KUKA KRL program: EPS_2_251349_MH87A_A_20250929014658.src

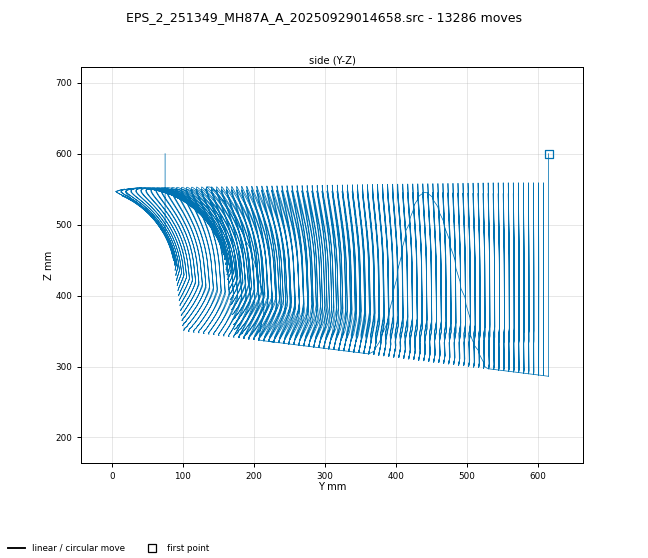
[picture p0: tool path of EPS_2_251349_MH87A_A_20250929014658.src, 13286 of 13288 moves have a stored position in this frame; points joined in program order, loops and branches not executed]
&ACCESS RVP
&REL 4
&COMMENT QRS 19112012
&PARAM EDITMASK = *
DEF PART()
EXT BAS (BAS_COMMAND :IN,REAL :IN )
INT I
BAS (#INITMOV,0 )

;KUKA QRS Post kuka4.cps  Date:22-06-2017 !

File_ID=2862

QRS_PRE_INIT()

;Init var - Until changes are made in qrs_pre_init
Outlet_Square_prg=0
Inlet_1_Square_prg=0
Inlet_2_Square_prg=0
Inlet_3_Square_prg=0
Inlet_4_Square_prg=0
Inlet_5_Square_prg=0

Outlet_1={X 0.000, Y 535.490, Z 458.500, B 0.000, E1 0.000 }
Inlet_1={X 0.000, Y 536.560, Z 443.500, B 0.000, E1 156.000 }
Outlet_1_type=201
Inlet_1_type=201
;QRS#1=Sidecore dimensions
;QRS#2=200-8" PVC SDR 35
;QRS#3=200-8" PVC SDR 35
;QRS#4=
;QRS#5=
;QRS#6=
;QRS#7=
;QRS#8=
;QRS#9=12-08 PSX
;QRS#10=12-08 PSX
;QRS#11=
;QRS#12=
;QRS#13=
;QRS#14=
;QRS#15=
;QRS#16=1220x127x838 2,75'
;QRS#17=EPS Height
;QRS#18=559
;QRS#19=*
;QRS#20= UPDATED VERSION 22-06-2017
;QRS#21=*
Outlet_Square=0100
Inlet_1_Square=0100
Inlet_2_Square=0
Inlet_3_Square=0
Inlet_4_Square=0
Inlet_5_Square=0
Mill_Square=1
Outlet_Square_Prg=204
Inlet_1_Square_prg=204

QRS_INIT()

$ADVANCE=5

; T1
PTP {E1 173.604,E2 173.604}
PTP {X 0,Y 615.51,A -85,B 0,C 180,E1 173.604,E2 173.604,E3 0,E4 0,E5 0,E6 0}
QRS_SPEED_INIT()
LIN {X 0,Y 615.51,Z 600,A -85,B 0,C 180,E1 173.604,E2 173.604,E3 0,E4 0,E5 0,E6 0} C_VEL
LIN {X 0,Y 615.51,Z 296.361,A -85,B 0,C 180,E1 173.604,E2 173.604} C_VEL
LIN {X 0,Y 615.51,Z 288.184,A -85,B 0,C 180,E1 173.604,E2 173.604} C_VEL
LIN {X 0,Y 615.494,Z 286.184,A -85,B 0,C 180,E1 173.418,E2 173.418} C_VEL
LIN {X 0,Y 615.499,Z 286.199,A -85,B 0,C 180,E1 170.801,E2 170.801} C_VEL
LIN {X 0,Y 615.469,Z 286.19,A -85,B 0,C 180,E1 168.139,E2 168.139} C_VEL
LIN {X 0,Y 615.478,Z 286.181,A -85,B 0,C 180,E1 165.451,E2 165.451} C_VEL
LIN {X 0,Y 615.488,Z 286.183,A -85,B 0,C 180,E1 162.729,E2 162.729} C_VEL
LIN {X 0,Y 615.491,Z 286.202,A -85,B 0,C 180,E1 159.967,E2 159.967} C_VEL
LIN {X 0,Y 615.48,Z 286.198,A -85,B 0,C 180,E1 157.656,E2 157.656} C_VEL
LIN {X 0,Y 615.46,Z 286.188,A -85,B 0,C 180,E1 155.007,E2 155.007} C_VEL
LIN {X 0,Y 615.459,Z 286.188,A -85,B 0,C 180,E1 152.821,E2 152.821} C_VEL
LIN {X 0,Y 615.478,Z 286.181,A -85,B 0,C 180,E1 150.207,E2 150.207} C_VEL
LIN {X 0,Y 615.487,Z 286.186,A -85,B 0,C 180,E1 147.542,E2 147.542} C_VEL
LIN {X 0,Y 615.487,Z 286.192,A -85,B 0,C 180,E1 145.185,E2 145.185} C_VEL
LIN {X 0,Y 615.491,Z 286.201,A -85,B 0,C 180,E1 142.758,E2 142.758} C_VEL
LIN {X 0,Y 615.474,Z 286.193,A -85,B 0,C 180,E1 140.249,E2 140.249} C_VEL
LIN {X 0,Y 615.456,Z 286.187,A -85,B 0,C 180,E1 137.644,E2 137.644} C_VEL
LIN {X 0,Y 615.473,Z 286.183,A -85,B 0,C 180,E1 134.93,E2 134.93} C_VEL
LIN {X 0,Y 615.498,Z 286.371,A -85,B 0,C 180,E1 134.036,E2 134.036} C_VEL
LIN {X 0,Y 615.487,Z 302.509,A -85,B 0,C 180,E1 131.474,E2 131.474} C_VEL
LIN {X 0,Y 615.461,Z 320.425,A -85,B 0,C 180,E1 128.697,E2 128.697} C_VEL
LIN {X 0,Y 615.464,Z 332.446,A -85,B 0,C 180,E1 126.871,E2 126.871} C_VEL
LIN {X 0,Y 615.462,Z 333.679,A -85,B 0,C 180,E1 126.807,E2 126.807} C_VEL
LIN {X 0,Y 615.496,Z 437.942,A -85,B 0,C 180,E1 125.565,E2 125.565} C_VEL
LIN {X 0,Y 615.494,Z 448.449,A -85,B 0,C 180,E1 125.364,E2 125.364} C_VEL
LIN {X 0,Y 615.497,Z 459.189,A -85,B 0,C 180,E1 125.064,E2 125.064} C_VEL
LIN {X 0,Y 615.499,Z 468.978,A -85,B 0,C 180,E1 124.702,E2 124.702} C_VEL
LIN {X 0,Y 615.478,Z 479.707,A -85,B 0,C 180,E1 124.192,E2 124.192} C_VEL
LIN {X 0,Y 615.49,Z 488.871,A -85,B 0,C 180,E1 123.656,E2 123.656} C_VEL
LIN {X 0,Y 615.499,Z 498.772,A -85,B 0,C 180,E1 122.943,E2 122.943} C_VEL
LIN {X 0,Y 615.495,Z 505.946,A -85,B 0,C 180,E1 122.332,E2 122.332} C_VEL
LIN {X 0,Y 615.494,Z 513.767,A -85,B 0,C 180,E1 121.535,E2 121.535} C_VEL
LIN {X 0,Y 615.497,Z 520.403,A -85,B 0,C 180,E1 120.729,E2 120.729} C_VEL
LIN {X 0,Y 615.486,Z 526.732,A -85,B 0,C 180,E1 119.794,E2 119.794} C_VEL
LIN {X 0,Y 615.492,Z 531.077,A -85,B 0,C 180,E1 119.031,E2 119.031} C_VEL
LIN {X 0,Y 615.49,Z 535.996,A -85,B 0,C 180,E1 117.915,E2 117.915} C_VEL
LIN {X 0,Y 615.486,Z 538.972,A -85,B 0,C 180,E1 117.045,E2 117.045} C_VEL
LIN {X 0,Y 615.495,Z 542.092,A -85,B 0,C 180,E1 115.57,E2 115.57} C_VEL
LIN {X 0,Y 615.495,Z 542.897,A -85,B 0,C 180,E1 114.991,E2 114.991} C_VEL
LIN {X 0,Y 615.493,Z 543.382,A -85,B 0,C 180,E1 114.009,E2 114.009} C_VEL
LIN {X 0,Y 615.485,Z 542.815,A -85,B 0,C 180,E1 112.845,E2 112.845} C_VEL
LIN {X 0,Y 615.496,Z 541.803,A -85,B 0,C 180,E1 112.136,E2 112.136} C_VEL
LIN {X 0,Y 615.491,Z 538.547,A -85,B 0,C 180,E1 110.731,E2 110.731} C_VEL
LIN {X 0,Y 615.49,Z 534.776,A -85,B 0,C 180,E1 109.685,E2 109.685} C_VEL
LIN {X 0,Y 615.496,Z 529.572,A -85,B 0,C 180,E1 108.607,E2 108.607} C_VEL
LIN {X 0,Y 615.491,Z 524.695,A -85,B 0,C 180,E1 107.785,E2 107.785} C_VEL
LIN {X 0,Y 615.493,Z 517.044,A -85,B 0,C 180,E1 106.757,E2 106.757} C_VEL
LIN {X 0,Y 615.5,Z 510.634,A -85,B 0,C 180,E1 106.037,E2 106.037} C_VEL
LIN {X 0,Y 615.497,Z 501.923,A -85,B 0,C 180,E1 105.226,E2 105.226} C_VEL
LIN {X 0,Y 615.49,Z 493.177,A -85,B 0,C 180,E1 104.549,E2 104.549} C_VEL
LIN {X 0,Y 615.487,Z 484.879,A -85,B 0,C 180,E1 104.008,E2 104.008} C_VEL
LIN {X 0,Y 615.485,Z 474.438,A -85,B 0,C 180,E1 103.453,E2 103.453} C_VEL
LIN {X 0,Y 615.498,Z 464.571,A -85,B 0,C 180,E1 103.033,E2 103.033} C_VEL
LIN {X 0,Y 615.498,Z 454.476,A -85,B 0,C 180,E1 102.697,E2 102.697} C_VEL
LIN {X 0,Y 615.497,Z 442.926,A -85,B 0,C 180,E1 102.425,E2 102.425} C_VEL
LIN {X 0,Y 615.497,Z 424.681,A -85,B 0,C 180,E1 102.174,E2 102.174} C_VEL
LIN {X 0,Y 615.49,Z 333.446,A -85,B 0,C 180,E1 101.098,E2 101.098} C_VEL
LIN {X 0,Y 615.491,Z 332.123,A -85,B 0,C 180,E1 101.003,E2 101.003} C_VEL
LIN {X 0,Y 615.474,Z 314.962,A -85,B 0,C 180,E1 98.371,E2 98.371} C_VEL
LIN {X 0,Y 615.488,Z 296.979,A -85,B 0,C 180,E1 95.57,E2 95.57} C_VEL
LIN {X 0,Y 615.497,Z 286.302,A -85,B 0,C 180,E1 93.846,E2 93.846} C_VEL
LIN {X 0,Y 615.493,Z 286.19,A -85,B 0,C 180,E1 91.309,E2 91.309} C_VEL
LIN {X 0,Y 615.478,Z 286.183,A -85,B 0,C 180,E1 88.691,E2 88.691} C_VEL
LIN {X 0,Y 615.472,Z 286.181,A -85,B 0,C 180,E1 86.071,E2 86.071} C_VEL
LIN {X 0,Y 615.49,Z 286.183,A -85,B 0,C 180,E1 83.42,E2 83.42} C_VEL
LIN {X 0,Y 615.494,Z 286.195,A -85,B 0,C 180,E1 80.801,E2 80.801} C_VEL
LIN {X 0,Y 615.496,Z 286.188,A -85,B 0,C 180,E1 78.139,E2 78.139} C_VEL
LIN {X 0,Y 615.472,Z 286.183,A -85,B 0,C 180,E1 75.45,E2 75.45} C_VEL
LIN {X 0,Y 615.472,Z 286.182,A -85,B 0,C 180,E1 72.729,E2 72.729} C_VEL
LIN {X 0,Y 615.493,Z 286.191,A -85,B 0,C 180,E1 69.967,E2 69.967} C_VEL
LIN {X 0,Y 615.49,Z 286.189,A -85,B 0,C 180,E1 67.155,E2 67.155} C_VEL
LIN {X 0,Y 615.463,Z 286.184,A -85,B 0,C 180,E1 64.436,E2 64.436} C_VEL
LIN {X 0,Y 615.463,Z 286.183,A -85,B 0,C 180,E1 62.084,E2 62.084} C_VEL
LIN {X 0,Y 615.463,Z 286.183,A -85,B 0,C 180,E1 59.838,E2 59.838} C_VEL
LIN {X 0,Y 615.461,Z 286.184,A -85,B 0,C 180,E1 57.541,E2 57.541} C_VEL
LIN {X 0,Y 615.472,Z 286.183,A -85,B 0,C 180,E1 55.184,E2 55.184} C_VEL
LIN {X 0,Y 615.486,Z 286.183,A -85,B 0,C 180,E1 52.758,E2 52.758} C_VEL
LIN {X 0,Y 615.497,Z 286.198,A -85,B 0,C 180,E1 49.91,E2 49.91} C_VEL
LIN {X 0,Y 615.494,Z 286.196,A -85,B 0,C 180,E1 47.647,E2 47.647} C_VEL
LIN {X 0,Y 615.467,Z 286.186,A -85,B 0,C 180,E1 44.929,E2 44.929} C_VEL
LIN {X 0,Y 615.456,Z 286.185,A -85,B 0,C 180,E1 42.356,E2 42.356} C_VEL
LIN {X 0,Y 615.474,Z 286.183,A -85,B 0,C 180,E1 39.751,E2 39.751} C_VEL
LIN {X 0,Y 615.491,Z 286.197,A -85,B 0,C 180,E1 36.937,E2 36.937} C_VEL
LIN {X 0,Y 615.465,Z 286.188,A -85,B 0,C 180,E1 34.023,E2 34.023} C_VEL
LIN {X 0,Y 615.456,Z 286.187,A -85,B 0,C 180,E1 31.687,E2 31.687} C_VEL
LIN {X 0,Y 615.452,Z 286.187,A -85,B 0,C 180,E1 29.408,E2 29.408} C_VEL
LIN {X 0,Y 615.45,Z 286.186,A -85,B 0,C 180,E1 27.038,E2 27.038} C_VEL
LIN {X 0,Y 615.448,Z 286.188,A -85,B 0,C 180,E1 24.994,E2 24.994} C_VEL
LIN {X 0,Y 615.449,Z 286.188,A -85,B 0,C 180,E1 22.846,E2 22.846} C_VEL
LIN {X 0,Y 615.447,Z 286.187,A -85,B 0,C 180,E1 20.546,E2 20.546} C_VEL
LIN {X 0,Y 615.452,Z 286.189,A -85,B 0,C 180,E1 18.594,E2 18.594} C_VEL
LIN {X 0,Y 615.452,Z 286.189,A -85,B 0,C 180,E1 16.419,E2 16.419} C_VEL
LIN {X 0,Y 615.444,Z 286.187,A -85,B 0,C 180,E1 13.875,E2 13.875} C_VEL
LIN {X 0,Y 615.473,Z 286.185,A -85,B 0,C 180,E1 11.193,E2 11.193} C_VEL
LIN {X 0,Y 615.495,Z 286.192,A -85,B 0,C 180,E1 8.537,E2 8.537} C_VEL
LIN {X 0,Y 615.485,Z 286.194,A -85,B 0,C 180,E1 5.899,E2 5.899} C_VEL
LIN {X 0,Y 615.446,Z 286.191,A -85,B 0,C 180,E1 3.273,E2 3.273} C_VEL
LIN {X 0,Y 615.457,Z 286.194,A -85,B 0,C 180,E1 1.309,E2 1.309} C_VEL
LIN {X 0,Y 615.437,Z 286.19,A -85,B 0,C 180,E1 -1.309,E2 -1.309} C_VEL
LIN {X 0,Y 615.443,Z 286.192,A -85,B 0,C 180,E1 -3.273,E2 -3.273} C_VEL
LIN {X 0,Y 615.459,Z 286.194,A -85,B 0,C 180,E1 -5.241,E2 -5.241} C_VEL
LIN {X 0,Y 615.482,Z 286.196,A -85,B 0,C 180,E1 -7.216,E2 -7.216} C_VEL
LIN {X 0,Y 615.439,Z 286.193,A -85,B 0,C 180,E1 -9.863,E2 -9.863} C_VEL
LIN {X 0,Y 615.451,Z 286.194,A -85,B 0,C 180,E1 -11.861,E2 -11.861} C_VEL
LIN {X 0,Y 615.462,Z 286.196,A -85,B 0,C 180,E1 -13.922,E2 -13.922} C_VEL
LIN {X 0,Y 615.43,Z 286.192,A -85,B 0,C 180,E1 -16.588,E2 -16.588} C_VEL
LIN {X 0,Y 615.433,Z 286.194,A -85,B 0,C 180,E1 -18.647,E2 -18.647} C_VEL
LIN {X 0,Y 615.434,Z 286.196,A -85,B 0,C 180,E1 -20.732,E2 -20.732} C_VEL
LIN {X 0,Y 615.442,Z 286.196,A -85,B 0,C 180,E1 -22.846,E2 -22.846} C_VEL
LIN {X 0,Y 615.445,Z 286.196,A -85,B 0,C 180,E1 -24.993,E2 -24.993} C_VEL
LIN {X 0,Y 615.443,Z 286.197,A -85,B 0,C 180,E1 -27.179,E2 -27.179} C_VEL
LIN {X 0,Y 615.442,Z 286.196,A -85,B 0,C 180,E1 -29.408,E2 -29.408} C_VEL
LIN {X 0,Y 615.435,Z 286.195,A -85,B 0,C 180,E1 -31.688,E2 -31.688} C_VEL
LIN {X 0,Y 615.428,Z 286.194,A -85,B 0,C 180,E1 -34.025,E2 -34.025} C_VEL
LIN {X 0,Y 615.424,Z 286.193,A -85,B 0,C 180,E1 -36.429,E2 -36.429} C_VEL
LIN {X 0,Y 615.443,Z 286.189,A -85,B 0,C 180,E1 -39.057,E2 -39.057} C_VEL
LIN {X 0,Y 615.464,Z 286.188,A -85,B 0,C 180,E1 -41.475,E2 -41.475} C_VEL
LIN {X 0,Y 615.497,Z 286.195,A -85,B 0,C 180,E1 -44.148,E2 -44.148} C_VEL
LIN {X 0,Y 615.439,Z 286.196,A -85,B 0,C 180,E1 -46.957,E2 -46.957} C_VEL
LIN {X 0,Y 615.426,Z 286.194,A -85,B 0,C 180,E1 -49.388,E2 -49.388} C_VEL
LIN {X 0,Y 615.465,Z 286.198,A -85,B 0,C 180,E1 -51.094,E2 -51.094} C_VEL
LIN {X 0,Y 615.436,Z 286.196,A -85,B 0,C 180,E1 -53.572,E2 -53.572} C_VEL
LIN {X 0,Y 615.425,Z 286.195,A -85,B 0,C 180,E1 -55.974,E2 -55.974} C_VEL
LIN {X 0,Y 615.421,Z 286.194,A -85,B 0,C 180,E1 -58.311,E2 -58.311} C_VEL
LIN {X 0,Y 615.421,Z 286.193,A -85,B 0,C 180,E1 -60.59,E2 -60.59} C_VEL
LIN {X 0,Y 615.421,Z 286.193,A -85,B 0,C 180,E1 -62.82,E2 -62.82} C_VEL
LIN {X 0,Y 615.419,Z 286.193,A -85,B 0,C 180,E1 -65.005,E2 -65.005} C_VEL
LIN {X 0,Y 615.42,Z 286.193,A -85,B 0,C 180,E1 -67.153,E2 -67.153} C_VEL
LIN {X 0,Y 615.495,Z 286.312,A -85,B 0,C 180,E1 -68.436,E2 -68.436} C_VEL
LIN {X 0,Y 615.496,Z 289.294,A -85,B 0,C 180,E1 -68.919,E2 -68.919} C_VEL
LIN {X 0,Y 615.478,Z 308.747,A -85,B 0,C 180,E1 -71.724,E2 -71.724} C_VEL
LIN {X 0,Y 615.487,Z 330.234,A -85,B 0,C 180,E1 -74.774,E2 -74.774} C_VEL
LIN {X 0,Y 615.471,Z 346.94,A -85,B 0,C 180,E1 -77.092,E2 -77.092} C_VEL
LIN {X 0,Y 615.465,Z 348.891,A -85,B 0,C 180,E1 -77.155,E2 -77.155} C_VEL
LIN {X 0,Y 615.498,Z 452.932,A -85,B 0,C 180,E1 -78.39,E2 -78.39} C_VEL
LIN {X 0,Y 615.498,Z 462.101,A -85,B 0,C 180,E1 -78.557,E2 -78.557} C_VEL
LIN {X 0,Y 615.498,Z 473.92,A -85,B 0,C 180,E1 -78.882,E2 -78.882} C_VEL
LIN {X 0,Y 615.496,Z 484.795,A -85,B 0,C 180,E1 -79.29,E2 -79.29} C_VEL
LIN {X 0,Y 615.475,Z 493.986,A -85,B 0,C 180,E1 -79.722,E2 -79.722} C_VEL
LIN {X 0,Y 615.476,Z 503.936,A -85,B 0,C 180,E1 -80.304,E2 -80.304} C_VEL
LIN {X 0,Y 615.497,Z 513.22,A -85,B 0,C 180,E1 -80.967,E2 -80.967} C_VEL
LIN {X 0,Y 615.497,Z 521.002,A -85,B 0,C 180,E1 -81.629,E2 -81.629} C_VEL
LIN {X 0,Y 615.494,Z 529.063,A -85,B 0,C 180,E1 -82.454,E2 -82.454} C_VEL
LIN {X 0,Y 615.497,Z 535.609,A -85,B 0,C 180,E1 -83.255,E2 -83.255} C_VEL
LIN {X 0,Y 615.488,Z 541.389,A -85,B 0,C 180,E1 -84.101,E2 -84.101} C_VEL
LIN {X 0,Y 615.492,Z 546.829,A -85,B 0,C 180,E1 -85.087,E2 -85.087} C_VEL
LIN {X 0,Y 615.488,Z 551.104,A -85,B 0,C 180,E1 -86.071,E2 -86.071} C_VEL
LIN {X 0,Y 615.488,Z 553.378,A -85,B 0,C 180,E1 -86.727,E2 -86.727} C_VEL
LIN {X 0,Y 615.49,Z 556.601,A -85,B 0,C 180,E1 -88.037,E2 -88.037} C_VEL
LIN {X 0,Y 615.489,Z 558.102,A -85,B 0,C 180,E1 -89.346,E2 -89.346} C_VEL
LIN {X 0,Y 615.488,Z 558.39,A -85,B 0,C 180,E1 -90,E2 -90} C_VEL
LIN {X 0,Y 615.484,Z 557.532,A -85,B 0,C 180,E1 -91.309,E2 -91.309} C_VEL
LIN {X 0,Y 615.49,Z 556.602,A -85,B 0,C 180,E1 -91.963,E2 -91.963} C_VEL
LIN {X 0,Y 615.488,Z 553.378,A -85,B 0,C 180,E1 -93.273,E2 -93.273} C_VEL
LIN {X 0,Y 615.496,Z 549.839,A -85,B 0,C 180,E1 -94.256,E2 -94.256} C_VEL
LIN {X 0,Y 615.488,Z 545.195,A -85,B 0,C 180,E1 -95.241,E2 -95.241} C_VEL
LIN {X 0,Y 615.495,Z 539.286,A -85,B 0,C 180,E1 -96.227,E2 -96.227} C_VEL
LIN {X 0,Y 615.49,Z 533.24,A -85,B 0,C 180,E1 -97.059,E2 -97.059} C_VEL
LIN {X 0,Y 615.491,Z 526.073,A -85,B 0,C 180,E1 -97.876,E2 -97.876} C_VEL
LIN {X 0,Y 615.496,Z 517.257,A -85,B 0,C 180,E1 -98.702,E2 -98.702} C_VEL
LIN {X 0,Y 615.494,Z 508.785,A -85,B 0,C 180,E1 -99.364,E2 -99.364} C_VEL
LIN {X 0,Y 615.468,Z 499.914,A -85,B 0,C 180,E1 -99.945,E2 -99.945} C_VEL
LIN {X 0,Y 615.486,Z 490.725,A -85,B 0,C 180,E1 -100.444,E2 -100.444} C_VEL
LIN {X 0,Y 615.497,Z 479.29,A -85,B 0,C 180,E1 -100.932,E2 -100.932} C_VEL
LIN {X 0,Y 615.497,Z 468.733,A -85,B 0,C 180,E1 -101.276,E2 -101.276} C_VEL
LIN {X 0,Y 615.497,Z 456.832,A -85,B 0,C 180,E1 -101.547,E2 -101.547} C_VEL
LIN {X 0,Y 615.488,Z 440.015,A -85,B 0,C 180,E1 -101.777,E2 -101.777} C_VEL
LIN {X 0,Y 615.467,Z 347.736,A -85,B 0,C 180,E1 -102.866,E2 -102.866} C_VEL
LIN {X 0,Y 615.473,Z 346.52,A -85,B 0,C 180,E1 -102.95,E2 -102.95} C_VEL
LIN {X 0,Y 615.491,Z 326.62,A -85,B 0,C 180,E1 -105.735,E2 -105.735} C_VEL
LIN {X 0,Y 615.463,Z 307.634,A -85,B 0,C 180,E1 -108.436,E2 -108.436} C_VEL
LIN {X 0,Y 615.494,Z 289.295,A -85,B 0,C 180,E1 -111.081,E2 -111.081} C_VEL
LIN {X 0,Y 615.495,Z 286.312,A -85,B 0,C 180,E1 -111.563,E2 -111.563} C_VEL
LIN {X 0,Y 615.477,Z 286.188,A -85,B 0,C 180,E1 -114.272,E2 -114.272} C_VEL
LIN {X 0,Y 615.432,Z 286.191,A -85,B 0,C 180,E1 -117.036,E2 -117.036} C_VEL
LIN {X 0,Y 615.433,Z 286.192,A -85,B 0,C 180,E1 -119.409,E2 -119.409} C_VEL
LIN {X 0,Y 615.436,Z 286.193,A -85,B 0,C 180,E1 -121.688,E2 -121.688} C_VEL
LIN {X 0,Y 615.446,Z 286.194,A -85,B 0,C 180,E1 -124.025,E2 -124.025} C_VEL
LIN {X 0,Y 615.495,Z 286.192,A -85,B 0,C 180,E1 -126.938,E2 -126.938} C_VEL
LIN {X 0,Y 615.472,Z 286.183,A -85,B 0,C 180,E1 -129.751,E2 -129.751} C_VEL
LIN {X 0,Y 615.451,Z 286.188,A -85,B 0,C 180,E1 -132.356,E2 -132.356} C_VEL
LIN {X 0,Y 615.469,Z 286.197,A -85,B 0,C 180,E1 -135.07,E2 -135.07} C_VEL
LIN {X 0,Y 615.495,Z 286.186,A -85,B 0,C 180,E1 -137.919,E2 -137.919} C_VEL
LIN {X 0,Y 615.497,Z 286.181,A -85,B 0,C 180,E1 -140.251,E2 -140.251} C_VEL
LIN {X 0,Y 615.468,Z 286.183,A -85,B 0,C 180,E1 -143.066,E2 -143.066} C_VEL
LIN {X 0,Y 615.468,Z 286.184,A -85,B 0,C 180,E1 -145.302,E2 -145.302} C_VEL
LIN {X 0,Y 615.464,Z 286.189,A -85,B 0,C 180,E1 -147.673,E2 -147.673} C_VEL
LIN {X 0,Y 615.48,Z 286.196,A -85,B 0,C 180,E1 -150.207,E2 -150.207} C_VEL
LIN {X 0,Y 615.489,Z 286.189,A -85,B 0,C 180,E1 -152.955,E2 -152.955} C_VEL
LIN {X 0,Y 615.495,Z 286.177,A -85,B 0,C 180,E1 -155.729,E2 -155.729} C_VEL
LIN {X 0,Y 615.477,Z 286.188,A -85,B 0,C 180,E1 -158.568,E2 -158.568} C_VEL
LIN {X 0,Y 615.487,Z 286.197,A -85,B 0,C 180,E1 -161.354,E2 -161.354} C_VEL
LIN {X 0,Y 615.486,Z 286.181,A -85,B 0,C 180,E1 -164.095,E2 -164.095} C_VEL
LIN {X 0,Y 615.496,Z 286.177,A -85,B 0,C 180,E1 -166.799,E2 -166.799} C_VEL
LIN {X 0,Y 615.484,Z 286.19,A -85,B 0,C 180,E1 -169.473,E2 -169.473} C_VEL
LIN {X 0,Y 615.49,Z 286.197,A -85,B 0,C 180,E1 -172.125,E2 -172.125} C_VEL
LIN {X 0,Y 615.48,Z 286.185,A -85,B 0,C 180,E1 -174.759,E2 -174.759} C_VEL
LIN {X 0,Y 615.492,Z 286.177,A -85,B 0,C 180,E1 -177.382,E2 -177.382} C_VEL
LIN {X 0,Y 615.492,Z 286.182,A -85,B 0,C 180,E1 -180,E2 -180} C_VEL
LIN {X 0,Y 615.491,Z 286.196,A -85,B 0,C 180,E1 -182.618,E2 -182.618} C_VEL
LIN {X 0,Y 615.478,Z 286.193,A -85,B 0,C 180,E1 -185.241,E2 -185.241} C_VEL
LIN {X 0,Y 615.494,Z 286.184,A -85,B 0,C 180,E1 -186.582,E2 -186.582} C_VEL
LIN {X 0,Y 614.817,Z 286.342,A -85,B 0,C 180,E1 -187.128,E2 -187.128} C_VEL
LIN {X 0,Y 611.988,Z 286.745,A -85,B 0,C 180,E1 -188.014,E2 -188.014} C_VEL
LIN {X 0,Y 609.597,Z 287.063,A -85,B 0,C 180,E1 -188.727,E2 -188.727} C_VEL
LIN {X 0,Y 608.556,Z 287.185,A -85,B 0,C 180,E1 -189.276,E2 -189.276} C_VEL
LIN {X 0,Y 608.462,Z 287.192,A -85,B 0,C 180,E1 -189.462,E2 -189.462} C_VEL
LIN {X 0,Y 608.451,Z 287.188,A -85,B 0,C 180,E1 -192,E2 -192} C_VEL
LIN {X 0,Y 608.471,Z 287.183,A -85,B 0,C 180,E1 -194.721,E2 -194.721} C_VEL
LIN {X 0,Y 608.455,Z 287.19,A -85,B 0,C 180,E1 -197.477,E2 -197.477} C_VEL
LIN {X 0,Y 608.455,Z 287.193,A -85,B 0,C 180,E1 -200.275,E2 -200.275} C_VEL
LIN {X 0,Y 608.461,Z 287.191,A -85,B 0,C 180,E1 -202.476,E2 -202.476} C_VEL
LIN {X 0,Y 608.448,Z 287.194,A -85,B 0,C 180,E1 -204.571,E2 -204.571} C_VEL
LIN {X 0,Y 608.437,Z 287.188,A -85,B 0,C 180,E1 -207.199,E2 -207.199} C_VEL
LIN {X 0,Y 608.463,Z 287.184,A -85,B 0,C 180,E1 -209.78,E2 -209.78} C_VEL
LIN {X 0,Y 608.462,Z 287.189,A -85,B 0,C 180,E1 -212.522,E2 -212.522} C_VEL
LIN {X 0,Y 608.428,Z 287.198,A -85,B 0,C 180,E1 -215.279,E2 -215.279} C_VEL
LIN {X 0,Y 608.451,Z 287.189,A -85,B 0,C 180,E1 -217.748,E2 -217.748} C_VEL
LIN {X 0,Y 608.433,Z 287.188,A -85,B 0,C 180,E1 -220.327,E2 -220.327} C_VEL
LIN {X 0,Y 608.448,Z 287.187,A -85,B 0,C 180,E1 -222.96,E2 -222.96} C_VEL
LIN {X 0,Y 608.491,Z 287.335,A -85,B 0,C 180,E1 -225.876,E2 -225.876} C_VEL
LIN {X 0,Y 608.517,Z 302.67,A -85,B 0,C 180,E1 -228.333,E2 -228.333} C_VEL
LIN {X 0,Y 608.464,Z 320.072,A -85,B 0,C 180,E1 -231.057,E2 -231.057} C_VEL
LIN {X 0,Y 608.477,Z 332.845,A -85,B 0,C 180,E1 -233.006,E2 -233.006} C_VEL
LIN {X 0,Y 608.552,Z 335.969,A -85,B 0,C 180,E1 -233.076,E2 -233.076} C_VEL
LIN {X 0,Y 608.547,Z 438.665,A -85,B 0,C 180,E1 -234.31,E2 -234.31} C_VEL
LIN {X 0,Y 608.537,Z 448.438,A -85,B 0,C 180,E1 -234.5,E2 -234.5} C_VEL
LIN {X 0,Y 608.547,Z 458.602,A -85,B 0,C 180,E1 -234.783,E2 -234.783} C_VEL
LIN {X 0,Y 608.522,Z 469.459,A -85,B 0,C 180,E1 -235.189,E2 -235.189} C_VEL
LIN {X 0,Y 608.48,Z 478.865,A -85,B 0,C 180,E1 -235.632,E2 -235.632} C_VEL
LIN {X 0,Y 608.48,Z 489.549,A -85,B 0,C 180,E1 -236.264,E2 -236.264} C_VEL
LIN {X 0,Y 608.477,Z 498.683,A -85,B 0,C 180,E1 -236.924,E2 -236.924} C_VEL
LIN {X 0,Y 608.455,Z 507.454,A -85,B 0,C 180,E1 -237.69,E2 -237.69} C_VEL
LIN {X 0,Y 608.456,Z 515.069,A -85,B 0,C 180,E1 -238.489,E2 -238.489} C_VEL
LIN {X 0,Y 608.464,Z 521.294,A -85,B 0,C 180,E1 -239.263,E2 -239.263} C_VEL
LIN {X 0,Y 608.436,Z 527.646,A -85,B 0,C 180,E1 -240.219,E2 -240.219} C_VEL
LIN {X 0,Y 608.427,Z 531.881,A -85,B 0,C 180,E1 -240.978,E2 -240.978} C_VEL
LIN {X 0,Y 608.435,Z 536.768,A -85,B 0,C 180,E1 -242.108,E2 -242.108} C_VEL
LIN {X 0,Y 608.429,Z 539.167,A -85,B 0,C 180,E1 -242.802,E2 -242.802} C_VEL
LIN {X 0,Y 608.426,Z 542.039,A -85,B 0,C 180,E1 -243.964,E2 -243.964} C_VEL
LIN {X 0,Y 608.438,Z 543.102,A -85,B 0,C 180,E1 -244.698,E2 -244.698} C_VEL
LIN {X 0,Y 608.435,Z 543.973,A -85,B 0,C 180,E1 -246.154,E2 -246.154} C_VEL
LIN {X 0,Y 608.422,Z 543.634,A -85,B 0,C 180,E1 -246.875,E2 -246.875} C_VEL
LIN {X 0,Y 608.425,Z 541.637,A -85,B 0,C 180,E1 -248.307,E2 -248.307} C_VEL
LIN {X 0,Y 608.436,Z 539.025,A -85,B 0,C 180,E1 -249.329,E2 -249.329} C_VEL
LIN {X 0,Y 608.422,Z 535.003,A -85,B 0,C 180,E1 -250.428,E2 -250.428} C_VEL
LIN {X 0,Y 608.432,Z 530.963,A -85,B 0,C 180,E1 -251.295,E2 -251.295} C_VEL
LIN {X 0,Y 608.448,Z 524.672,A -85,B 0,C 180,E1 -252.35,E2 -252.35} C_VEL
LIN {X 0,Y 608.458,Z 518.35,A -85,B 0,C 180,E1 -253.216,E2 -253.216} C_VEL
LIN {X 0,Y 608.462,Z 510.718,A -85,B 0,C 180,E1 -254.078,E2 -254.078} C_VEL
LIN {X 0,Y 608.468,Z 502.488,A -85,B 0,C 180,E1 -254.851,E2 -254.851} C_VEL
LIN {X 0,Y 608.474,Z 493.756,A -85,B 0,C 180,E1 -255.536,E2 -255.536} C_VEL
LIN {X 0,Y 608.483,Z 484.611,A -85,B 0,C 180,E1 -256.133,E2 -256.133} C_VEL
LIN {X 0,Y 608.494,Z 475.129,A -85,B 0,C 180,E1 -256.644,E2 -256.644} C_VEL
LIN {X 0,Y 608.54,Z 464.162,A -85,B 0,C 180,E1 -257.112,E2 -257.112} C_VEL
LIN {X 0,Y 608.544,Z 453.027,A -85,B 0,C 180,E1 -257.473,E2 -257.473} C_VEL
LIN {X 0,Y 608.553,Z 441.897,A -85,B 0,C 180,E1 -257.727,E2 -257.727} C_VEL
LIN {X 0,Y 608.562,Z 425.004,A -85,B 0,C 180,E1 -257.96,E2 -257.96} C_VEL
LIN {X 0,Y 608.535,Z 333.32,A -85,B 0,C 180,E1 -259.056,E2 -259.056} C_VEL
LIN {X 0,Y 608.477,Z 331.914,A -85,B 0,C 180,E1 -259.199,E2 -259.199} C_VEL
LIN {X 0,Y 608.473,Z 313.659,A -85,B 0,C 180,E1 -262.033,E2 -262.033} C_VEL
LIN {X 0,Y 608.498,Z 297.768,A -85,B 0,C 180,E1 -264.532,E2 -264.532} C_VEL
LIN {X 0,Y 608.487,Z 287.286,A -85,B 0,C 180,E1 -266.234,E2 -266.234} C_VEL
LIN {X 0,Y 608.477,Z 287.189,A -85,B 0,C 180,E1 -268.676,E2 -268.676} C_VEL
LIN {X 0,Y 608.463,Z 287.185,A -85,B 0,C 180,E1 -271.324,E2 -271.324} C_VEL
LIN {X 0,Y 608.443,Z 287.186,A -85,B 0,C 180,E1 -273.974,E2 -273.974} C_VEL
LIN {X 0,Y 608.48,Z 287.185,A -85,B 0,C 180,E1 -276.633,E2 -276.633} C_VEL
LIN {X 0,Y 608.478,Z 287.194,A -85,B 0,C 180,E1 -279.306,E2 -279.306} C_VEL
LIN {X 0,Y 608.465,Z 287.188,A -85,B 0,C 180,E1 -282,E2 -282} C_VEL
LIN {X 0,Y 608.465,Z 287.183,A -85,B 0,C 180,E1 -284.721,E2 -284.721} C_VEL
LIN {X 0,Y 608.446,Z 287.188,A -85,B 0,C 180,E1 -287.477,E2 -287.477} C_VEL
LIN {X 0,Y 608.469,Z 287.195,A -85,B 0,C 180,E1 -290.274,E2 -290.274} C_VEL
LIN {X 0,Y 608.445,Z 287.188,A -85,B 0,C 180,E1 -293.124,E2 -293.124} C_VEL
LIN {X 0,Y 608.452,Z 287.185,A -85,B 0,C 180,E1 -295.717,E2 -295.717} C_VEL
LIN {X 0,Y 608.446,Z 287.186,A -85,B 0,C 180,E1 -298.267,E2 -298.267} C_VEL
LIN {X 0,Y 608.446,Z 287.187,A -85,B 0,C 180,E1 -300.546,E2 -300.546} C_VEL
LIN {X 0,Y 608.451,Z 287.188,A -85,B 0,C 180,E1 -302.88,E2 -302.88} C_VEL
LIN {X 0,Y 608.445,Z 287.191,A -85,B 0,C 180,E1 -305.278,E2 -305.278} C_VEL
LIN {X 0,Y 608.471,Z 287.188,A -85,B 0,C 180,E1 -308.241,E2 -308.241} C_VEL
LIN {X 0,Y 608.445,Z 287.186,A -85,B 0,C 180,E1 -311.34,E2 -311.34} C_VEL
LIN {X 0,Y 608.46,Z 287.194,A -85,B 0,C 180,E1 -314.264,E2 -314.264} C_VEL
LIN {X 0,Y 608.449,Z 287.19,A -85,B 0,C 180,E1 -317.04,E2 -317.04} C_VEL
LIN {X 0,Y 608.455,Z 287.185,A -85,B 0,C 180,E1 -319.697,E2 -319.697} C_VEL
LIN {X 0,Y 608.483,Z 287.187,A -85,B 0,C 180,E1 -322.84,E2 -322.84} C_VEL
LIN {X 0,Y 608.47,Z 287.193,A -85,B 0,C 180,E1 -325.531,E2 -325.531} C_VEL
LIN {X 0,Y 608.465,Z 287.189,A -85,B 0,C 180,E1 -327.905,E2 -327.905} C_VEL
LIN {X 0,Y 608.461,Z 287.188,A -85,B 0,C 180,E1 -330.22,E2 -330.22} C_VEL
LIN {X 0,Y 608.43,Z 287.188,A -85,B 0,C 180,E1 -332.802,E2 -332.802} C_VEL
LIN {X 0,Y 608.434,Z 287.19,A -85,B 0,C 180,E1 -334.698,E2 -334.698} C_VEL
LIN {X 0,Y 608.434,Z 287.19,A -85,B 0,C 180,E1 -336.875,E2 -336.875} C_VEL
LIN {X 0,Y 608.438,Z 287.187,A -85,B 0,C 180,E1 -339.329,E2 -339.329} C_VEL
LIN {X 0,Y 608.42,Z 287.188,A -85,B 0,C 180,E1 -341.827,E2 -341.827} C_VEL
LIN {X 0,Y 608.467,Z 287.187,A -85,B 0,C 180,E1 -344.594,E2 -344.594} C_VEL
LIN {X 0,Y 608.478,Z 287.195,A -85,B 0,C 180,E1 -347.323,E2 -347.323} C_VEL
LIN {X 0,Y 608.43,Z 287.191,A -85,B 0,C 180,E1 -350.022,E2 -350.022} C_VEL
LIN {X 0,Y 608.42,Z 287.188,A -85,B 0,C 180,E1 -352.7,E2 -352.7} C_VEL
LIN {X 0,Y 608.438,Z 287.188,A -85,B 0,C 180,E1 -355.362,E2 -355.362} C_VEL
LIN {X 0,Y 608.464,Z 287.192,A -85,B 0,C 180,E1 -358.014,E2 -358.014} C_VEL
LIN {X 0,Y 608.474,Z 287.191,A -85,B 0,C 180,E1 -360.662,E2 -360.662} C_VEL
LIN {X 0,Y 608.413,Z 287.191,A -85,B 0,C 180,E1 -363.311,E2 -363.311} C_VEL
LIN {X 0,Y 608.438,Z 287.191,A -85,B 0,C 180,E1 -365.302,E2 -365.302} C_VEL
LIN {X 0,Y 608.443,Z 287.193,A -85,B 0,C 180,E1 -367.299,E2 -367.299} C_VEL
LIN {X 0,Y 608.414,Z 287.191,A -85,B 0,C 180,E1 -369.978,E2 -369.978} C_VEL
LIN {X 0,Y 608.428,Z 287.19,A -85,B 0,C 180,E1 -372,E2 -372} C_VEL
LIN {X 0,Y 608.423,Z 287.193,A -85,B 0,C 180,E1 -374.038,E2 -374.038} C_VEL
LIN {X 0,Y 608.404,Z 287.192,A -85,B 0,C 180,E1 -376.508,E2 -376.508} C_VEL
LIN {X 0,Y 608.427,Z 287.188,A -85,B 0,C 180,E1 -378.87,E2 -378.87} C_VEL
LIN {X 0,Y 608.445,Z 287.188,A -85,B 0,C 180,E1 -381.692,E2 -381.692} C_VEL
LIN {X 0,Y 608.443,Z 287.199,A -85,B 0,C 180,E1 -384.571,E2 -384.571} C_VEL
LIN {X 0,Y 608.41,Z 287.191,A -85,B 0,C 180,E1 -387.52,E2 -387.52} C_VEL
LIN {X 0,Y 608.413,Z 287.19,A -85,B 0,C 180,E1 -389.782,E2 -389.782} C_VEL
LIN {X 0,Y 608.424,Z 287.189,A -85,B 0,C 180,E1 -392.516,E2 -392.516} C_VEL
LIN {X 0,Y 608.432,Z 287.196,A -85,B 0,C 180,E1 -395.278,E2 -395.278} C_VEL
LIN {X 0,Y 608.451,Z 287.198,A -85,B 0,C 180,E1 -397.747,E2 -397.747} C_VEL
LIN {X 0,Y 608.432,Z 287.192,A -85,B 0,C 180,E1 -400.327,E2 -400.327} C_VEL
LIN {X 0,Y 608.435,Z 287.195,A -85,B 0,C 180,E1 -402.331,E2 -402.331} C_VEL
LIN {X 0,Y 608.412,Z 287.194,A -85,B 0,C 180,E1 -404.8,E2 -404.8} C_VEL
LIN {X 0,Y 608.406,Z 287.194,A -85,B 0,C 180,E1 -407.036,E2 -407.036} C_VEL
LIN {X 0,Y 608.441,Z 287.196,A -85,B 0,C 180,E1 -408.822,E2 -408.822} C_VEL
LIN {X 0,Y 608.406,Z 287.194,A -85,B 0,C 180,E1 -411.407,E2 -411.407} C_VEL
LIN {X 0,Y 608.453,Z 287.197,A -85,B 0,C 180,E1 -413.085,E2 -413.085} C_VEL
LIN {X 0,Y 608.452,Z 287.192,A -85,B 0,C 180,E1 -415.529,E2 -415.529} C_VEL
LIN {X 0,Y 608.433,Z 287.192,A -85,B 0,C 180,E1 -417.903,E2 -417.903} C_VEL
LIN {X 0,Y 608.419,Z 287.192,A -85,B 0,C 180,E1 -420.218,E2 -420.218} C_VEL
LIN {X 0,Y 608.412,Z 287.192,A -85,B 0,C 180,E1 -422.48,E2 -422.48} C_VEL
LIN {X 0,Y 608.395,Z 287.194,A -85,B 0,C 180,E1 -424.696,E2 -424.696} C_VEL
LIN {X 0,Y 608.408,Z 287.194,A -85,B 0,C 180,E1 -426.874,E2 -426.874} C_VEL
LIN {X 0,Y 608.509,Z 287.349,A -85,B 0,C 180,E1 -428.354,E2 -428.354} C_VEL
LIN {X 0,Y 608.5,Z 302.577,A -85,B 0,C 180,E1 -430.606,E2 -430.606} C_VEL
LIN {X 0,Y 608.471,Z 319.469,A -85,B 0,C 180,E1 -433.043,E2 -433.043} C_VEL
LIN {X 0,Y 608.443,Z 336.362,A -85,B 0,C 180,E1 -435.45,E2 -435.45} C_VEL
LIN {X 0,Y 608.497,Z 347.291,A -85,B 0,C 180,E1 -436.963,E2 -436.963} C_VEL
LIN {X 0,Y 608.559,Z 354.288,A -85,B 0,C 180,E1 -437.07,E2 -437.07} C_VEL
LIN {X 0,Y 608.551,Z 453.06,A -85,B 0,C 180,E1 -438.255,E2 -438.255} C_VEL
LIN {X 0,Y 608.55,Z 463.042,A -85,B 0,C 180,E1 -438.445,E2 -438.445} C_VEL
LIN {X 0,Y 608.537,Z 473.729,A -85,B 0,C 180,E1 -438.742,E2 -438.742} C_VEL
LIN {X 0,Y 608.511,Z 484.938,A -85,B 0,C 180,E1 -439.165,E2 -439.165} C_VEL
LIN {X 0,Y 608.493,Z 494.151,A -85,B 0,C 180,E1 -439.603,E2 -439.603} C_VEL
LIN {X 0,Y 608.462,Z 504.139,A -85,B 0,C 180,E1 -440.191,E2 -440.191} C_VEL
LIN {X 0,Y 608.471,Z 513.47,A -85,B 0,C 180,E1 -440.862,E2 -440.862} C_VEL
LIN {X 0,Y 608.485,Z 521.295,A -85,B 0,C 180,E1 -441.532,E2 -441.532} C_VEL
LIN {X 0,Y 608.469,Z 529.41,A -85,B 0,C 180,E1 -442.367,E2 -442.367} C_VEL
LIN {X 0,Y 608.458,Z 536.174,A -85,B 0,C 180,E1 -443.201,E2 -443.201} C_VEL
LIN {X 0,Y 608.429,Z 541.834,A -85,B 0,C 180,E1 -444.033,E2 -444.033} C_VEL
LIN {X 0,Y 608.432,Z 547.324,A -85,B 0,C 180,E1 -445.03,E2 -445.03} C_VEL
LIN {X 0,Y 608.428,Z 551.641,A -85,B 0,C 180,E1 -446.026,E2 -446.026} C_VEL
LIN {X 0,Y 608.419,Z 553.932,A -85,B 0,C 180,E1 -446.689,E2 -446.689} C_VEL
LIN {X 0,Y 608.435,Z 557.194,A -85,B 0,C 180,E1 -448.014,E2 -448.014} C_VEL
LIN {X 0,Y 608.432,Z 558.713,A -85,B 0,C 180,E1 -449.338,E2 -449.338} C_VEL
LIN {X 0,Y 608.428,Z 559,A -85,B 0,C 180,E1 -450,E2 -450} C_VEL
LIN {X 0,Y 608.436,Z 558.134,A -85,B 0,C 180,E1 -451.324,E2 -451.324} C_VEL
LIN {X 0,Y 608.435,Z 557.194,A -85,B 0,C 180,E1 -451.986,E2 -451.986} C_VEL
LIN {X 0,Y 608.419,Z 553.933,A -85,B 0,C 180,E1 -453.311,E2 -453.311} C_VEL
LIN {X 0,Y 608.44,Z 550.357,A -85,B 0,C 180,E1 -454.306,E2 -454.306} C_VEL
LIN {X 0,Y 608.454,Z 545.666,A -85,B 0,C 180,E1 -455.302,E2 -455.302} C_VEL
LIN {X 0,Y 608.449,Z 539.707,A -85,B 0,C 180,E1 -456.3,E2 -456.3} C_VEL
LIN {X 0,Y 608.46,Z 533.677,A -85,B 0,C 180,E1 -457.133,E2 -457.133} C_VEL
LIN {X 0,Y 608.456,Z 526.393,A -85,B 0,C 180,E1 -457.967,E2 -457.967} C_VEL
LIN {X 0,Y 608.475,Z 517.526,A -85,B 0,C 180,E1 -458.803,E2 -458.803} C_VEL
LIN {X 0,Y 608.476,Z 509.011,A -85,B 0,C 180,E1 -459.473,E2 -459.473} C_VEL
LIN {X 0,Y 608.488,Z 500.098,A -85,B 0,C 180,E1 -460.061,E2 -460.061} C_VEL
LIN {X 0,Y 608.517,Z 490.883,A -85,B 0,C 180,E1 -460.565,E2 -460.565} C_VEL
LIN {X 0,Y 608.525,Z 479.268,A -85,B 0,C 180,E1 -461.064,E2 -461.064} C_VEL
LIN {X 0,Y 608.546,Z 468.026,A -85,B 0,C 180,E1 -461.428,E2 -461.428} C_VEL
LIN {X 0,Y 608.556,Z 456.965,A -85,B 0,C 180,E1 -461.681,E2 -461.681} C_VEL
LIN {X 0,Y 608.544,Z 440.158,A -85,B 0,C 180,E1 -461.914,E2 -461.914} C_VEL
LIN {X 0,Y 608.515,Z 347.748,A -85,B 0,C 180,E1 -463.015,E2 -463.015} C_VEL
LIN {X 0,Y 608.467,Z 346.651,A -85,B 0,C 180,E1 -463.101,E2 -463.101} C_VEL
LIN {X 0,Y 608.481,Z 325.504,A -85,B 0,C 180,E1 -466.093,E2 -466.093} C_VEL
LIN {X 0,Y 608.492,Z 307.204,A -85,B 0,C 180,E1 -468.723,E2 -468.723} C_VEL
LIN {X 0,Y 608.57,Z 289.305,A -85,B 0,C 180,E1 -471.332,E2 -471.332} C_VEL
LIN {X 0,Y 608.488,Z 287.264,A -85,B 0,C 180,E1 -471.691,E2 -471.691} C_VEL
LIN {X 0,Y 608.426,Z 287.19,A -85,B 0,C 180,E1 -474.572,E2 -474.572} C_VEL
LIN {X 0,Y 608.412,Z 287.191,A -85,B 0,C 180,E1 -477.196,E2 -477.196} C_VEL
LIN {X 0,Y 608.413,Z 287.19,A -85,B 0,C 180,E1 -479.023,E2 -479.023} C_VEL
LIN {X 0,Y 608.429,Z 287.188,A -85,B 0,C 180,E1 -481.319,E2 -481.319} C_VEL
LIN {X 0,Y 608.421,Z 287.19,A -85,B 0,C 180,E1 -483.728,E2 -483.728} C_VEL
LIN {X 0,Y 608.432,Z 287.19,A -85,B 0,C 180,E1 -486.093,E2 -486.093} C_VEL
LIN {X 0,Y 608.43,Z 287.195,A -85,B 0,C 180,E1 -488.591,E2 -488.591} C_VEL
LIN {X 0,Y 608.472,Z 287.189,A -85,B 0,C 180,E1 -491.344,E2 -491.344} C_VEL
LIN {X 0,Y 608.469,Z 287.185,A -85,B 0,C 180,E1 -493.87,E2 -493.87} C_VEL
LIN {X 0,Y 608.448,Z 287.187,A -85,B 0,C 180,E1 -496.693,E2 -496.693} C_VEL
LIN {X 0,Y 608.431,Z 287.189,A -85,B 0,C 180,E1 -498.822,E2 -498.822} C_VEL
LIN {X 0,Y 608.47,Z 287.195,A -85,B 0,C 180,E1 -501.76,E2 -501.76} C_VEL
LIN {X 0,Y 608.461,Z 287.197,A -85,B 0,C 180,E1 -503.953,E2 -503.953} C_VEL
LIN {X 0,Y 608.466,Z 287.192,A -85,B 0,C 180,E1 -506.33,E2 -506.33} C_VEL
LIN {X 0,Y 608.48,Z 287.186,A -85,B 0,C 180,E1 -508.727,E2 -508.727} C_VEL
LIN {X 0,Y 608.477,Z 287.182,A -85,B 0,C 180,E1 -511.38,E2 -511.38} C_VEL
LIN {X 0,Y 608.444,Z 287.187,A -85,B 0,C 180,E1 -513.965,E2 -513.965} C_VEL
LIN {X 0,Y 608.464,Z 287.185,A -85,B 0,C 180,E1 -516.155,E2 -516.155} C_VEL
LIN {X 0,Y 608.467,Z 287.185,A -85,B 0,C 180,E1 -518.309,E2 -518.309} C_VEL
LIN {X 0,Y 608.456,Z 287.196,A -85,B 0,C 180,E1 -521.131,E2 -521.131} C_VEL
LIN {X 0,Y 608.461,Z 287.187,A -85,B 0,C 180,E1 -523.906,E2 -523.906} C_VEL
LIN {X 0,Y 608.471,Z 287.183,A -85,B 0,C 180,E1 -526.644,E2 -526.644} C_VEL
LIN {X 0,Y 608.465,Z 287.188,A -85,B 0,C 180,E1 -529.35,E2 -529.35} C_VEL
LIN {X 0,Y 608.481,Z 287.194,A -85,B 0,C 180,E1 -532.033,E2 -532.033} C_VEL
LIN {X 0,Y 608.461,Z 287.187,A -85,B 0,C 180,E1 -534.698,E2 -534.698} C_VEL
LIN {X 0,Y 608.482,Z 287.181,A -85,B 0,C 180,E1 -537.352,E2 -537.352} C_VEL
LIN {X 0,Y 608.482,Z 287.184,A -85,B 0,C 180,E1 -540,E2 -540} C_VEL
LIN {X 0,Y 608.481,Z 287.192,A -85,B 0,C 180,E1 -542.648,E2 -542.648} C_VEL
LIN {X 0,Y 608.459,Z 287.19,A -85,B 0,C 180,E1 -545.302,E2 -545.302} C_VEL
LIN {X 0,Y 608.473,Z 287.183,A -85,B 0,C 180,E1 -547.967,E2 -547.967} C_VEL
LIN {X 0,Y 608.462,Z 287.192,A -85,B 0,C 180,E1 -549.462,E2 -549.462} C_VEL
LIN {X 0,Y 607.771,Z 287.273,A -85,B 0,C 180,E1 -550.015,E2 -550.015} C_VEL
LIN {X 0,Y 604.91,Z 287.631,A -85,B 0,C 180,E1 -550.912,E2 -550.912} C_VEL
LIN {X 0,Y 602.511,Z 287.933,A -85,B 0,C 180,E1 -551.634,E2 -551.634} C_VEL
LIN {X 0,Y 601.488,Z 288.054,A -85,B 0,C 180,E1 -552.19,E2 -552.19} C_VEL
LIN {X 0,Y 601.408,Z 288.063,A -85,B 0,C 180,E1 -552.379,E2 -552.379} C_VEL
LIN {X 0,Y 601.428,Z 288.061,A -85,B 0,C 180,E1 -554.897,E2 -554.897} C_VEL
LIN {X 0,Y 601.399,Z 288.073,A -85,B 0,C 180,E1 -557.688,E2 -557.688} C_VEL
LIN {X 0,Y 601.419,Z 288.065,A -85,B 0,C 180,E1 -560.522,E2 -560.522} C_VEL
LIN {X 0,Y 601.395,Z 288.065,A -85,B 0,C 180,E1 -563.411,E2 -563.411} C_VEL
LIN {X 0,Y 601.42,Z 288.064,A -85,B 0,C 180,E1 -565.868,E2 -565.868} C_VEL
LIN {X 0,Y 601.43,Z 288.07,A -85,B 0,C 180,E1 -568.787,E2 -568.787} C_VEL
LIN {X 0,Y 601.415,Z 288.064,A -85,B 0,C 180,E1 -571.454,E2 -571.454} C_VEL
LIN {X 0,Y 601.419,Z 288.061,A -85,B 0,C 180,E1 -574.119,E2 -574.119} C_VEL
LIN {X 0,Y 601.436,Z 288.07,A -85,B 0,C 180,E1 -577.382,E2 -577.382} C_VEL
LIN {X 0,Y 601.403,Z 288.067,A -85,B 0,C 180,E1 -579.996,E2 -579.996} C_VEL
LIN {X 0,Y 601.385,Z 288.066,A -85,B 0,C 180,E1 -582.673,E2 -582.673} C_VEL
LIN {X 0,Y 601.398,Z 288.068,A -85,B 0,C 180,E1 -584.533,E2 -584.533} C_VEL
LIN {X 0,Y 601.457,Z 288.27,A -85,B 0,C 180,E1 -585.788,E2 -585.788} C_VEL
LIN {X 0,Y 601.493,Z 300.778,A -85,B 0,C 180,E1 -587.817,E2 -587.817} C_VEL
LIN {X 0,Y 601.462,Z 317.433,A -85,B 0,C 180,E1 -590.462,E2 -590.462} C_VEL
LIN {X 0,Y 601.431,Z 332.698,A -85,B 0,C 180,E1 -592.838,E2 -592.838} C_VEL
LIN {X 0,Y 601.648,Z 334.924,A -85,B 0,C 180,E1 -592.912,E2 -592.912} C_VEL
LIN {X 0,Y 601.615,Z 438.524,A -85,B 0,C 180,E1 -594.171,E2 -594.171} C_VEL
LIN {X 0,Y 601.585,Z 448.456,A -85,B 0,C 180,E1 -594.365,E2 -594.365} C_VEL
LIN {X 0,Y 601.576,Z 458.34,A -85,B 0,C 180,E1 -594.641,E2 -594.641} C_VEL
LIN {X 0,Y 601.53,Z 469.785,A -85,B 0,C 180,E1 -595.076,E2 -595.076} C_VEL
LIN {X 0,Y 601.491,Z 480.138,A -85,B 0,C 180,E1 -595.582,E2 -595.582} C_VEL
LIN {X 0,Y 601.479,Z 489.18,A -85,B 0,C 180,E1 -596.123,E2 -596.123} C_VEL
LIN {X 0,Y 601.476,Z 497.148,A -85,B 0,C 180,E1 -596.69,E2 -596.69} C_VEL
LIN {X 0,Y 601.442,Z 506.377,A -85,B 0,C 180,E1 -597.485,E2 -597.485} C_VEL
LIN {X 0,Y 601.393,Z 513.999,A -85,B 0,C 180,E1 -598.273,E2 -598.273} C_VEL
LIN {X 0,Y 601.381,Z 520.412,A -85,B 0,C 180,E1 -599.056,E2 -599.056} C_VEL
LIN {X 0,Y 601.375,Z 527.074,A -85,B 0,C 180,E1 -600.049,E2 -600.049} C_VEL
LIN {X 0,Y 601.333,Z 531.994,A -85,B 0,C 180,E1 -600.943,E2 -600.943} C_VEL
LIN {X 0,Y 601.376,Z 535.635,A -85,B 0,C 180,E1 -601.751,E2 -601.751} C_VEL
LIN {X 0,Y 601.328,Z 539.535,A -85,B 0,C 180,E1 -602.883,E2 -602.883} C_VEL
LIN {X 0,Y 601.335,Z 542.353,A -85,B 0,C 180,E1 -604.148,E2 -604.148} C_VEL
LIN {X 0,Y 601.326,Z 543.593,A -85,B 0,C 180,E1 -605.118,E2 -605.118} C_VEL
LIN {X 0,Y 601.343,Z 543.936,A -85,B 0,C 180,E1 -605.855,E2 -605.855} C_VEL
LIN {X 0,Y 601.32,Z 543.235,A -85,B 0,C 180,E1 -607.313,E2 -607.313} C_VEL
LIN {X 0,Y 601.342,Z 542.216,A -85,B 0,C 180,E1 -608.038,E2 -608.038} C_VEL
LIN {X 0,Y 601.337,Z 539.483,A -85,B 0,C 180,E1 -609.225,E2 -609.225} C_VEL
LIN {X 0,Y 601.328,Z 536.224,A -85,B 0,C 180,E1 -610.188,E2 -610.188} C_VEL
LIN {X 0,Y 601.363,Z 530.726,A -85,B 0,C 180,E1 -611.399,E2 -611.399} C_VEL
LIN {X 0,Y 601.388,Z 524.233,A -85,B 0,C 180,E1 -612.487,E2 -612.487} C_VEL
LIN {X 0,Y 601.394,Z 516.807,A -85,B 0,C 180,E1 -613.484,E2 -613.484} C_VEL
LIN {X 0,Y 601.403,Z 510.102,A -85,B 0,C 180,E1 -614.235,E2 -614.235} C_VEL
LIN {X 0,Y 601.419,Z 502.798,A -85,B 0,C 180,E1 -614.93,E2 -614.93} C_VEL
LIN {X 0,Y 601.465,Z 494.112,A -85,B 0,C 180,E1 -615.623,E2 -615.623} C_VEL
LIN {X 0,Y 601.47,Z 485.269,A -85,B 0,C 180,E1 -616.215,E2 -616.215} C_VEL
LIN {X 0,Y 601.509,Z 475.666,A -85,B 0,C 180,E1 -616.744,E2 -616.744} C_VEL
LIN {X 0,Y 601.56,Z 464.861,A -85,B 0,C 180,E1 -617.218,E2 -617.218} C_VEL
LIN {X 0,Y 601.601,Z 453.11,A -85,B 0,C 180,E1 -617.604,E2 -617.604} C_VEL
LIN {X 0,Y 601.604,Z 442.06,A -85,B 0,C 180,E1 -617.861,E2 -617.861} C_VEL
LIN {X 0,Y 601.643,Z 425.141,A -85,B 0,C 180,E1 -618.097,E2 -618.097} C_VEL
LIN {X 0,Y 601.52,Z 333.583,A -85,B 0,C 180,E1 -619.202,E2 -619.202} C_VEL
LIN {X 0,Y 601.445,Z 332.236,A -85,B 0,C 180,E1 -619.31,E2 -619.31} C_VEL
LIN {X 0,Y 601.452,Z 314.394,A -85,B 0,C 180,E1 -622.108,E2 -622.108} C_VEL
LIN {X 0,Y 601.525,Z 297.454,A -85,B 0,C 180,E1 -624.805,E2 -624.805} C_VEL
LIN {X 0,Y 601.462,Z 288.164,A -85,B 0,C 180,E1 -626.336,E2 -626.336} C_VEL
LIN {X 0,Y 601.442,Z 288.059,A -85,B 0,C 180,E1 -629.331,E2 -629.331} C_VEL
LIN {X 0,Y 601.423,Z 288.062,A -85,B 0,C 180,E1 -632.009,E2 -632.009} C_VEL
LIN {X 0,Y 601.429,Z 288.067,A -85,B 0,C 180,E1 -634.692,E2 -634.692} C_VEL
LIN {X 0,Y 601.445,Z 288.066,A -85,B 0,C 180,E1 -637.385,E2 -637.385} C_VEL
LIN {X 0,Y 601.436,Z 288.06,A -85,B 0,C 180,E1 -640.095,E2 -640.095} C_VEL
LIN {X 0,Y 601.414,Z 288.062,A -85,B 0,C 180,E1 -642.828,E2 -642.828} C_VEL
LIN {X 0,Y 601.415,Z 288.068,A -85,B 0,C 180,E1 -645.591,E2 -645.591} C_VEL
LIN {X 0,Y 601.427,Z 288.067,A -85,B 0,C 180,E1 -648.392,E2 -648.392} C_VEL
LIN {X 0,Y 601.404,Z 288.063,A -85,B 0,C 180,E1 -651.24,E2 -651.24} C_VEL
LIN {X 0,Y 601.459,Z 288.059,A -85,B 0,C 180,E1 -654.14,E2 -654.14} C_VEL
LIN {X 0,Y 601.417,Z 288.065,A -85,B 0,C 180,E1 -657.362,E2 -657.362} C_VEL
LIN {X 0,Y 601.417,Z 288.068,A -85,B 0,C 180,E1 -659.393,E2 -659.393} C_VEL
LIN {X 0,Y 601.408,Z 288.067,A -85,B 0,C 180,E1 -661.727,E2 -661.727} C_VEL
LIN {X 0,Y 601.425,Z 288.062,A -85,B 0,C 180,E1 -664.119,E2 -664.119} C_VEL
LIN {X 0,Y 601.394,Z 288.064,A -85,B 0,C 180,E1 -666.584,E2 -666.584} C_VEL
LIN {X 0,Y 601.398,Z 288.064,A -85,B 0,C 180,E1 -669.128,E2 -669.128} C_VEL
LIN {X 0,Y 601.425,Z 288.064,A -85,B 0,C 180,E1 -671.765,E2 -671.765} C_VEL
LIN {X 0,Y 601.427,Z 288.071,A -85,B 0,C 180,E1 -674.535,E2 -674.535} C_VEL
LIN {X 0,Y 601.386,Z 288.067,A -85,B 0,C 180,E1 -677.327,E2 -677.327} C_VEL
LIN {X 0,Y 601.404,Z 288.062,A -85,B 0,C 180,E1 -680.004,E2 -680.004} C_VEL
LIN {X 0,Y 601.437,Z 288.061,A -85,B 0,C 180,E1 -682.618,E2 -682.618} C_VEL
LIN {X 0,Y 601.414,Z 288.065,A -85,B 0,C 180,E1 -685.881,E2 -685.881} C_VEL
LIN {X 0,Y 601.415,Z 288.061,A -85,B 0,C 180,E1 -688.547,E2 -688.547} C_VEL
LIN {X 0,Y 601.429,Z 288.062,A -85,B 0,C 180,E1 -691.373,E2 -691.373} C_VEL
LIN {X 0,Y 601.42,Z 288.069,A -85,B 0,C 180,E1 -694.382,E2 -694.382} C_VEL
LIN {X 0,Y 601.394,Z 288.072,A -85,B 0,C 180,E1 -696.589,E2 -696.589} C_VEL
LIN {X 0,Y 601.405,Z 288.062,A -85,B 0,C 180,E1 -699.477,E2 -699.477} C_VEL
LIN {X 0,Y 601.382,Z 288.065,A -85,B 0,C 180,E1 -701.607,E2 -701.607} C_VEL
LIN {X 0,Y 601.403,Z 288.064,A -85,B 0,C 180,E1 -704.408,E2 -704.408} C_VEL
LIN {X 0,Y 601.422,Z 288.071,A -85,B 0,C 180,E1 -707.172,E2 -707.172} C_VEL
LIN {X 0,Y 601.396,Z 288.069,A -85,B 0,C 180,E1 -709.904,E2 -709.904} C_VEL
LIN {X 0,Y 601.374,Z 288.066,A -85,B 0,C 180,E1 -712.614,E2 -712.614} C_VEL
LIN {X 0,Y 601.405,Z 288.063,A -85,B 0,C 180,E1 -715.308,E2 -715.308} C_VEL
LIN {X 0,Y 601.432,Z 288.067,A -85,B 0,C 180,E1 -717.991,E2 -717.991} C_VEL
LIN {X 0,Y 601.445,Z 288.066,A -85,B 0,C 180,E1 -720.669,E2 -720.669} C_VEL
LIN {X 0,Y 601.366,Z 288.068,A -85,B 0,C 180,E1 -723.35,E2 -723.35} C_VEL
LIN {X 0,Y 601.401,Z 288.066,A -85,B 0,C 180,E1 -725.364,E2 -725.364} C_VEL
LIN {X 0,Y 601.401,Z 288.069,A -85,B 0,C 180,E1 -727.385,E2 -727.385} C_VEL
LIN {X 0,Y 601.378,Z 288.067,A -85,B 0,C 180,E1 -730.096,E2 -730.096} C_VEL
LIN {X 0,Y 601.384,Z 288.066,A -85,B 0,C 180,E1 -732.143,E2 -732.143} C_VEL
LIN {X 0,Y 601.378,Z 288.068,A -85,B 0,C 180,E1 -734.206,E2 -734.206} C_VEL
LIN {X 0,Y 601.373,Z 288.067,A -85,B 0,C 180,E1 -736.604,E2 -736.604} C_VEL
LIN {X 0,Y 601.4,Z 288.063,A -85,B 0,C 180,E1 -739.099,E2 -739.099} C_VEL
LIN {X 0,Y 601.402,Z 288.068,A -85,B 0,C 180,E1 -741.959,E2 -741.959} C_VEL
LIN {X 0,Y 601.434,Z 288.066,A -85,B 0,C 180,E1 -744.291,E2 -744.291} C_VEL
LIN {X 0,Y 601.372,Z 288.069,A -85,B 0,C 180,E1 -747.354,E2 -747.354} C_VEL
LIN {X 0,Y 601.374,Z 288.071,A -85,B 0,C 180,E1 -749.395,E2 -749.395} C_VEL
LIN {X 0,Y 601.378,Z 288.068,A -85,B 0,C 180,E1 -751.728,E2 -751.728} C_VEL
LIN {X 0,Y 601.396,Z 288.065,A -85,B 0,C 180,E1 -754.12,E2 -754.12} C_VEL
LIN {X 0,Y 601.378,Z 288.066,A -85,B 0,C 180,E1 -756.584,E2 -756.584} C_VEL
LIN {X 0,Y 601.383,Z 288.067,A -85,B 0,C 180,E1 -759.128,E2 -759.128} C_VEL
LIN {X 0,Y 601.418,Z 288.068,A -85,B 0,C 180,E1 -761.765,E2 -761.765} C_VEL
LIN {X 0,Y 601.397,Z 288.072,A -85,B 0,C 180,E1 -764.532,E2 -764.532} C_VEL
LIN {X 0,Y 601.35,Z 288.07,A -85,B 0,C 180,E1 -767.324,E2 -767.324} C_VEL
LIN {X 0,Y 601.381,Z 288.067,A -85,B 0,C 180,E1 -769.43,E2 -769.43} C_VEL
LIN {X 0,Y 601.349,Z 288.07,A -85,B 0,C 180,E1 -771.726,E2 -771.726} C_VEL
LIN {X 0,Y 601.368,Z 288.069,A -85,B 0,C 180,E1 -773.743,E2 -773.743} C_VEL
LIN {X 0,Y 601.399,Z 288.064,A -85,B 0,C 180,E1 -776.069,E2 -776.069} C_VEL
LIN {X 0,Y 601.383,Z 288.066,A -85,B 0,C 180,E1 -778.551,E2 -778.551} C_VEL
LIN {X 0,Y 601.425,Z 288.065,A -85,B 0,C 180,E1 -781.373,E2 -781.373} C_VEL
LIN {X 0,Y 601.385,Z 288.072,A -85,B 0,C 180,E1 -784.38,E2 -784.38} C_VEL
LIN {X 0,Y 601.374,Z 288.075,A -85,B 0,C 180,E1 -786.588,E2 -786.588} C_VEL
LIN {X 0,Y 601.459,Z 288.241,A -85,B 0,C 180,E1 -788.223,E2 -788.223} C_VEL
LIN {X 0,Y 601.605,Z 295.089,A -85,B 0,C 180,E1 -789.269,E2 -789.269} C_VEL
LIN {X 0,Y 601.532,Z 315.85,A -85,B 0,C 180,E1 -792.316,E2 -792.316} C_VEL
LIN {X 0,Y 601.454,Z 335.156,A -85,B 0,C 180,E1 -795.104,E2 -795.104} C_VEL
LIN {X 0,Y 601.476,Z 347.285,A -85,B 0,C 180,E1 -796.808,E2 -796.808} C_VEL
LIN {X 0,Y 601.641,Z 350.711,A -85,B 0,C 180,E1 -796.876,E2 -796.876} C_VEL
LIN {X 0,Y 601.622,Z 453.059,A -85,B 0,C 180,E1 -798.118,E2 -798.118} C_VEL
LIN {X 0,Y 601.601,Z 463.044,A -85,B 0,C 180,E1 -798.31,E2 -798.31} C_VEL
LIN {X 0,Y 601.572,Z 473.867,A -85,B 0,C 180,E1 -798.615,E2 -798.615} C_VEL
LIN {X 0,Y 601.521,Z 484.943,A -85,B 0,C 180,E1 -799.038,E2 -799.038} C_VEL
LIN {X 0,Y 601.484,Z 495.641,A -85,B 0,C 180,E1 -799.566,E2 -799.566} C_VEL
LIN {X 0,Y 601.463,Z 504.141,A -85,B 0,C 180,E1 -800.075,E2 -800.075} C_VEL
LIN {X 0,Y 601.431,Z 513.471,A -85,B 0,C 180,E1 -800.754,E2 -800.754} C_VEL
LIN {X 0,Y 601.42,Z 521.294,A -85,B 0,C 180,E1 -801.431,E2 -801.431} C_VEL
LIN {X 0,Y 601.39,Z 529.411,A -85,B 0,C 180,E1 -802.276,E2 -802.276} C_VEL
LIN {X 0,Y 601.383,Z 536.175,A -85,B 0,C 180,E1 -803.12,E2 -803.12} C_VEL
LIN {X 0,Y 601.353,Z 541.835,A -85,B 0,C 180,E1 -803.962,E2 -803.962} C_VEL
LIN {X 0,Y 601.34,Z 547.324,A -85,B 0,C 180,E1 -804.971,E2 -804.971} C_VEL
LIN {X 0,Y 601.341,Z 551.642,A -85,B 0,C 180,E1 -805.979,E2 -805.979} C_VEL
LIN {X 0,Y 601.338,Z 553.933,A -85,B 0,C 180,E1 -806.65,E2 -806.65} C_VEL
LIN {X 0,Y 601.334,Z 557.192,A -85,B 0,C 180,E1 -807.991,E2 -807.991} C_VEL
LIN {X 0,Y 601.332,Z 558.713,A -85,B 0,C 180,E1 -809.33,E2 -809.33} C_VEL
LIN {X 0,Y 601.329,Z 559,A -85,B 0,C 180,E1 -810,E2 -810} C_VEL
LIN {X 0,Y 601.336,Z 558.135,A -85,B 0,C 180,E1 -811.339,E2 -811.339} C_VEL
LIN {X 0,Y 601.334,Z 557.193,A -85,B 0,C 180,E1 -812.009,E2 -812.009} C_VEL
LIN {X 0,Y 601.338,Z 553.934,A -85,B 0,C 180,E1 -813.35,E2 -813.35} C_VEL
LIN {X 0,Y 601.353,Z 550.357,A -85,B 0,C 180,E1 -814.357,E2 -814.357} C_VEL
LIN {X 0,Y 601.366,Z 545.665,A -85,B 0,C 180,E1 -815.365,E2 -815.365} C_VEL
LIN {X 0,Y 601.368,Z 539.499,A -85,B 0,C 180,E1 -816.404,E2 -816.404} C_VEL
LIN {X 0,Y 601.383,Z 533.676,A -85,B 0,C 180,E1 -817.217,E2 -817.217} C_VEL
LIN {X 0,Y 601.403,Z 526.392,A -85,B 0,C 180,E1 -818.061,E2 -818.061} C_VEL
LIN {X 0,Y 601.441,Z 517.528,A -85,B 0,C 180,E1 -818.907,E2 -818.907} C_VEL
LIN {X 0,Y 601.468,Z 509.015,A -85,B 0,C 180,E1 -819.585,E2 -819.585} C_VEL
LIN {X 0,Y 601.48,Z 500.102,A -85,B 0,C 180,E1 -820.179,E2 -820.179} C_VEL
LIN {X 0,Y 601.524,Z 490.888,A -85,B 0,C 180,E1 -820.689,E2 -820.689} C_VEL
LIN {X 0,Y 601.562,Z 479.437,A -85,B 0,C 180,E1 -821.188,E2 -821.188} C_VEL
LIN {X 0,Y 601.588,Z 468.027,A -85,B 0,C 180,E1 -821.562,E2 -821.562} C_VEL
LIN {X 0,Y 601.622,Z 456.963,A -85,B 0,C 180,E1 -821.817,E2 -821.817} C_VEL
LIN {X 0,Y 601.617,Z 440.158,A -85,B 0,C 180,E1 -822.053,E2 -822.053} C_VEL
LIN {X 0,Y 601.493,Z 347.734,A -85,B 0,C 180,E1 -823.17,E2 -823.17} C_VEL
LIN {X 0,Y 601.472,Z 346.651,A -85,B 0,C 180,E1 -823.256,E2 -823.256} C_VEL
LIN {X 0,Y 601.497,Z 325.504,A -85,B 0,C 180,E1 -826.285,E2 -826.285} C_VEL
LIN {X 0,Y 601.508,Z 307.907,A -85,B 0,C 180,E1 -828.845,E2 -828.845} C_VEL
LIN {X 0,Y 601.646,Z 290.511,A -85,B 0,C 180,E1 -831.41,E2 -831.41} C_VEL
LIN {X 0,Y 601.442,Z 288.143,A -85,B 0,C 180,E1 -831.823,E2 -831.823} C_VEL
LIN {X 0,Y 601.433,Z 288.064,A -85,B 0,C 180,E1 -834.293,E2 -834.293} C_VEL
LIN {X 0,Y 601.376,Z 288.067,A -85,B 0,C 180,E1 -837.115,E2 -837.115} C_VEL
LIN {X 0,Y 601.379,Z 288.067,A -85,B 0,C 180,E1 -839.395,E2 -839.395} C_VEL
LIN {X 0,Y 601.39,Z 288.067,A -85,B 0,C 180,E1 -841.728,E2 -841.728} C_VEL
LIN {X 0,Y 601.409,Z 288.068,A -85,B 0,C 180,E1 -844.12,E2 -844.12} C_VEL
LIN {X 0,Y 601.435,Z 288.061,A -85,B 0,C 180,E1 -847.382,E2 -847.382} C_VEL
LIN {X 0,Y 601.39,Z 288.065,A -85,B 0,C 180,E1 -849.997,E2 -849.997} C_VEL
LIN {X 0,Y 601.379,Z 288.07,A -85,B 0,C 180,E1 -852.673,E2 -852.673} C_VEL
LIN {X 0,Y 601.396,Z 288.065,A -85,B 0,C 180,E1 -854.533,E2 -854.533} C_VEL
LIN {X 0,Y 601.41,Z 288.074,A -85,B 0,C 180,E1 -857.41,E2 -857.41} C_VEL
LIN {X 0,Y 601.401,Z 288.07,A -85,B 0,C 180,E1 -860.004,E2 -860.004} C_VEL
LIN {X 0,Y 601.435,Z 288.06,A -85,B 0,C 180,E1 -862.618,E2 -862.618} C_VEL
LIN {X 0,Y 601.427,Z 288.06,A -85,B 0,C 180,E1 -865.069,E2 -865.069} C_VEL
LIN {X 0,Y 601.415,Z 288.063,A -85,B 0,C 180,E1 -867.484,E2 -867.484} C_VEL
LIN {X 0,Y 601.427,Z 288.063,A -85,B 0,C 180,E1 -869.852,E2 -869.852} C_VEL
LIN {X 0,Y 601.417,Z 288.073,A -85,B 0,C 180,E1 -872.637,E2 -872.637} C_VEL
LIN {X 0,Y 601.405,Z 288.069,A -85,B 0,C 180,E1 -875.122,E2 -875.122} C_VEL
LIN {X 0,Y 601.417,Z 288.065,A -85,B 0,C 180,E1 -877.395,E2 -877.395} C_VEL
LIN {X 0,Y 601.407,Z 288.063,A -85,B 0,C 180,E1 -880.191,E2 -880.191} C_VEL
LIN {X 0,Y 601.434,Z 288.065,A -85,B 0,C 180,E1 -883.014,E2 -883.014} C_VEL
LIN {X 0,Y 601.423,Z 288.066,A -85,B 0,C 180,E1 -885.908,E2 -885.908} C_VEL
LIN {X 0,Y 601.438,Z 288.06,A -85,B 0,C 180,E1 -888.542,E2 -888.542} C_VEL
LIN {X 0,Y 601.44,Z 288.06,A -85,B 0,C 180,E1 -891.263,E2 -891.263} C_VEL
LIN {X 0,Y 601.423,Z 288.07,A -85,B 0,C 180,E1 -893.963,E2 -893.963} C_VEL
LIN {X 0,Y 601.425,Z 288.067,A -85,B 0,C 180,E1 -896.651,E2 -896.651} C_VEL
LIN {X 0,Y 601.452,Z 288.058,A -85,B 0,C 180,E1 -899.331,E2 -899.331} C_VEL
LIN {X 0,Y 601.43,Z 288.061,A -85,B 0,C 180,E1 -902.009,E2 -902.009} C_VEL
LIN {X 0,Y 601.428,Z 288.068,A -85,B 0,C 180,E1 -904.692,E2 -904.692} C_VEL
LIN {X 0,Y 601.442,Z 288.065,A -85,B 0,C 180,E1 -907.385,E2 -907.385} C_VEL
LIN {X 0,Y 601.427,Z 288.061,A -85,B 0,C 180,E1 -910.095,E2 -910.095} C_VEL
LIN {X 0,Y 601.408,Z 288.063,A -85,B 0,C 180,E1 -912.379,E2 -912.379} C_VEL
LIN {X 0,Y 600.749,Z 288.148,A -85,B 0,C 180,E1 -912.938,E2 -912.938} C_VEL
LIN {X 0,Y 597.9,Z 288.507,A -85,B 0,C 180,E1 -913.846,E2 -913.846} C_VEL
LIN {X 0,Y 595.486,Z 288.804,A -85,B 0,C 180,E1 -914.576,E2 -914.576} C_VEL
LIN {X 0,Y 594.447,Z 288.933,A -85,B 0,C 180,E1 -915.14,E2 -915.14} C_VEL
LIN {X 0,Y 594.36,Z 288.945,A -85,B 0,C 180,E1 -915.33,E2 -915.33} C_VEL
LIN {X 0,Y 594.378,Z 288.951,A -85,B 0,C 180,E1 -917.904,E2 -917.904} C_VEL
LIN {X 0,Y 594.37,Z 288.94,A -85,B 0,C 180,E1 -920.914,E2 -920.914} C_VEL
LIN {X 0,Y 594.38,Z 288.941,A -85,B 0,C 180,E1 -923.705,E2 -923.705} C_VEL
LIN {X 0,Y 594.392,Z 288.941,A -85,B 0,C 180,E1 -926.024,E2 -926.024} C_VEL
LIN {X 0,Y 594.378,Z 288.945,A -85,B 0,C 180,E1 -928.999,E2 -928.999} C_VEL
LIN {X 0,Y 594.374,Z 288.94,A -85,B 0,C 180,E1 -931.642,E2 -931.642} C_VEL
LIN {X 0,Y 594.377,Z 288.942,A -85,B 0,C 180,E1 -934.58,E2 -934.58} C_VEL
LIN {X 0,Y 594.386,Z 288.944,A -85,B 0,C 180,E1 -937.608,E2 -937.608} C_VEL
LIN {X 0,Y 594.361,Z 288.941,A -85,B 0,C 180,E1 -940.568,E2 -940.568} C_VEL
LIN {X 0,Y 594.374,Z 288.945,A -85,B 0,C 180,E1 -943.299,E2 -943.299} C_VEL
LIN {X 0,Y 594.411,Z 289.108,A -85,B 0,C 180,E1 -945.67,E2 -945.67} C_VEL
LIN {X 0,Y 594.554,Z 295.369,A -85,B 0,C 180,E1 -946.717,E2 -946.717} C_VEL
LIN {X 0,Y 594.481,Z 312.238,A -85,B 0,C 180,E1 -949.442,E2 -949.442} C_VEL
LIN {X 0,Y 594.407,Z 330.748,A -85,B 0,C 180,E1 -952.389,E2 -952.389} C_VEL
LIN {X 0,Y 594.442,Z 333.09,A -85,B 0,C 180,E1 -952.709,E2 -952.709} C_VEL
LIN {X 0,Y 594.739,Z 338.304,A -85,B 0,C 180,E1 -952.797,E2 -952.797} C_VEL
LIN {X 0,Y 594.676,Z 438.344,A -85,B 0,C 180,E1 -954.027,E2 -954.027} C_VEL
LIN {X 0,Y 594.64,Z 448.704,A -85,B 0,C 180,E1 -954.234,E2 -954.234} C_VEL
LIN {X 0,Y 594.604,Z 458.303,A -85,B 0,C 180,E1 -954.504,E2 -954.504} C_VEL
LIN {X 0,Y 594.562,Z 469.154,A -85,B 0,C 180,E1 -954.916,E2 -954.916} C_VEL
LIN {X 0,Y 594.499,Z 479.626,A -85,B 0,C 180,E1 -955.428,E2 -955.428} C_VEL
LIN {X 0,Y 594.451,Z 489.505,A -85,B 0,C 180,E1 -956.028,E2 -956.028} C_VEL
LIN {X 0,Y 594.426,Z 499.19,A -85,B 0,C 180,E1 -956.75,E2 -956.75} C_VEL
LIN {X 0,Y 594.395,Z 507.08,A -85,B 0,C 180,E1 -957.454,E2 -957.454} C_VEL
LIN {X 0,Y 594.344,Z 513.647,A -85,B 0,C 180,E1 -958.137,E2 -958.137} C_VEL
LIN {X 0,Y 594.3,Z 520.892,A -85,B 0,C 180,E1 -959.042,E2 -959.042} C_VEL
LIN {X 0,Y 594.288,Z 526.929,A -85,B 0,C 180,E1 -959.952,E2 -959.952} C_VEL
LIN {X 0,Y 594.254,Z 532.497,A -85,B 0,C 180,E1 -960.995,E2 -960.995} C_VEL
LIN {X 0,Y 594.277,Z 535.912,A -85,B 0,C 180,E1 -961.768,E2 -961.768} C_VEL
LIN {X 0,Y 594.23,Z 539.709,A -85,B 0,C 180,E1 -962.913,E2 -962.913} C_VEL
LIN {X 0,Y 594.229,Z 542.244,A -85,B 0,C 180,E1 -964.049,E2 -964.049} C_VEL
LIN {X 0,Y 594.218,Z 543.289,A -85,B 0,C 180,E1 -964.8,E2 -964.8} C_VEL
LIN {X 0,Y 594.211,Z 543.822,A -85,B 0,C 180,E1 -965.604,E2 -965.604} C_VEL
LIN {X 0,Y 594.217,Z 543.913,A -85,B 0,C 180,E1 -966.289,E2 -966.289} C_VEL
LIN {X 0,Y 594.243,Z 543.284,A -85,B 0,C 180,E1 -967.293,E2 -967.293} C_VEL
LIN {X 0,Y 594.229,Z 541.33,A -85,B 0,C 180,E1 -968.492,E2 -968.492} C_VEL
LIN {X 0,Y 594.268,Z 538.44,A -85,B 0,C 180,E1 -969.581,E2 -969.581} C_VEL
LIN {X 0,Y 594.258,Z 535.989,A -85,B 0,C 180,E1 -970.302,E2 -970.302} C_VEL
LIN {X 0,Y 594.285,Z 531.181,A -85,B 0,C 180,E1 -971.379,E2 -971.379} C_VEL
LIN {X 0,Y 594.309,Z 525.022,A -85,B 0,C 180,E1 -972.449,E2 -972.449} C_VEL
LIN {X 0,Y 594.328,Z 517.309,A -85,B 0,C 180,E1 -973.513,E2 -973.513} C_VEL
LIN {X 0,Y 594.342,Z 511.234,A -85,B 0,C 180,E1 -974.218,E2 -974.218} C_VEL
LIN {X 0,Y 594.411,Z 502.052,A -85,B 0,C 180,E1 -975.098,E2 -975.098} C_VEL
LIN {X 0,Y 594.434,Z 494.409,A -85,B 0,C 180,E1 -975.717,E2 -975.717} C_VEL
LIN {X 0,Y 594.458,Z 485.499,A -85,B 0,C 180,E1 -976.323,E2 -976.323} C_VEL
LIN {X 0,Y 594.522,Z 476.206,A -85,B 0,C 180,E1 -976.847,E2 -976.847} C_VEL
LIN {X 0,Y 594.589,Z 464.343,A -85,B 0,C 180,E1 -977.369,E2 -977.369} C_VEL
LIN {X 0,Y 594.658,Z 453.197,A -85,B 0,C 180,E1 -977.739,E2 -977.739} C_VEL
LIN {X 0,Y 594.66,Z 442.209,A -85,B 0,C 180,E1 -977.999,E2 -977.999} C_VEL
LIN {X 0,Y 594.709,Z 425.337,A -85,B 0,C 180,E1 -978.238,E2 -978.238} C_VEL
LIN {X 0,Y 594.674,Z 334.747,A -85,B 0,C 180,E1 -979.337,E2 -979.337} C_VEL
LIN {X 0,Y 594.414,Z 332.839,A -85,B 0,C 180,E1 -979.397,E2 -979.397} C_VEL
LIN {X 0,Y 594.426,Z 316.199,A -85,B 0,C 180,E1 -982.015,E2 -982.015} C_VEL
LIN {X 0,Y 594.503,Z 300.296,A -85,B 0,C 180,E1 -984.573,E2 -984.573} C_VEL
LIN {X 0,Y 594.469,Z 289.184,A -85,B 0,C 180,E1 -986.399,E2 -986.399} C_VEL
LIN {X 0,Y 594.402,Z 288.94,A -85,B 0,C 180,E1 -987.289,E2 -987.289} C_VEL
LIN {X 0,Y 594.416,Z 288.937,A -85,B 0,C 180,E1 -990,E2 -990} C_VEL
LIN {X 0,Y 594.411,Z 288.946,A -85,B 0,C 180,E1 -992.711,E2 -992.711} C_VEL
LIN {X 0,Y 594.395,Z 288.94,A -85,B 0,C 180,E1 -995.428,E2 -995.428} C_VEL
LIN {X 0,Y 594.397,Z 288.943,A -85,B 0,C 180,E1 -997.473,E2 -997.473} C_VEL
LIN {X 0,Y 594.394,Z 288.937,A -85,B 0,C 180,E1 -1000.216,E2 -1000.216} C_VEL
LIN {X 0,Y 594.365,Z 288.941,A -85,B 0,C 180,E1 -1002.983,E2 -1002.983} C_VEL
LIN {X 0,Y 594.37,Z 288.94,A -85,B 0,C 180,E1 -1005.078,E2 -1005.078} C_VEL
LIN {X 0,Y 594.378,Z 288.939,A -85,B 0,C 180,E1 -1007.194,E2 -1007.194} C_VEL
LIN {X 0,Y 594.377,Z 288.946,A -85,B 0,C 180,E1 -1010.054,E2 -1010.054} C_VEL
LIN {X 0,Y 594.358,Z 288.945,A -85,B 0,C 180,E1 -1012.968,E2 -1012.968} C_VEL
LIN {X 0,Y 594.364,Z 288.944,A -85,B 0,C 180,E1 -1015.194,E2 -1015.194} C_VEL
LIN {X 0,Y 594.388,Z 288.939,A -85,B 0,C 180,E1 -1017.527,E2 -1017.527} C_VEL
LIN {X 0,Y 594.372,Z 288.939,A -85,B 0,C 180,E1 -1020.326,E2 -1020.326} C_VEL
LIN {X 0,Y 594.377,Z 288.942,A -85,B 0,C 180,E1 -1022.95,E2 -1022.95} C_VEL
LIN {X 0,Y 594.352,Z 288.949,A -85,B 0,C 180,E1 -1025.409,E2 -1025.409} C_VEL
LIN {X 0,Y 594.388,Z 288.948,A -85,B 0,C 180,E1 -1027.941,E2 -1027.941} C_VEL
LIN {X 0,Y 594.369,Z 288.939,A -85,B 0,C 180,E1 -1030.821,E2 -1030.821} C_VEL
LIN {X 0,Y 594.352,Z 288.941,A -85,B 0,C 180,E1 -1033.301,E2 -1033.301} C_VEL
LIN {X 0,Y 594.363,Z 288.945,A -85,B 0,C 180,E1 -1036.161,E2 -1036.161} C_VEL
LIN {X 0,Y 594.377,Z 288.943,A -85,B 0,C 180,E1 -1039.178,E2 -1039.178} C_VEL
LIN {X 0,Y 594.375,Z 288.938,A -85,B 0,C 180,E1 -1042.058,E2 -1042.058} C_VEL
LIN {X 0,Y 594.352,Z 288.943,A -85,B 0,C 180,E1 -1044.677,E2 -1044.677} C_VEL
LIN {X 0,Y 594.381,Z 288.942,A -85,B 0,C 180,E1 -1047.089,E2 -1047.089} C_VEL
LIN {X 0,Y 594.388,Z 288.948,A -85,B 0,C 180,E1 -1049.672,E2 -1049.672} C_VEL
LIN {X 0,Y 594.341,Z 288.945,A -85,B 0,C 180,E1 -1052.537,E2 -1052.537} C_VEL
LIN {X 0,Y 594.364,Z 288.942,A -85,B 0,C 180,E1 -1054.806,E2 -1054.806} C_VEL
LIN {X 0,Y 594.354,Z 288.941,A -85,B 0,C 180,E1 -1057.268,E2 -1057.268} C_VEL
LIN {X 0,Y 594.363,Z 288.94,A -85,B 0,C 180,E1 -1059.946,E2 -1059.946} C_VEL
LIN {X 0,Y 594.377,Z 288.947,A -85,B 0,C 180,E1 -1062.806,E2 -1062.806} C_VEL
LIN {X 0,Y 594.364,Z 288.941,A -85,B 0,C 180,E1 -1065.837,E2 -1065.837} C_VEL
LIN {X 0,Y 594.375,Z 288.938,A -85,B 0,C 180,E1 -1068.404,E2 -1068.404} C_VEL
LIN {X 0,Y 594.377,Z 288.941,A -85,B 0,C 180,E1 -1071.158,E2 -1071.158} C_VEL
LIN {X 0,Y 594.366,Z 288.951,A -85,B 0,C 180,E1 -1073.891,E2 -1073.891} C_VEL
LIN {X 0,Y 594.328,Z 288.947,A -85,B 0,C 180,E1 -1076.61,E2 -1076.61} C_VEL
LIN {X 0,Y 594.356,Z 288.946,A -85,B 0,C 180,E1 -1078.645,E2 -1078.645} C_VEL
LIN {X 0,Y 594.417,Z 288.941,A -85,B 0,C 180,E1 -1080.677,E2 -1080.677} C_VEL
LIN {X 0,Y 594.32,Z 288.945,A -85,B 0,C 180,E1 -1083.389,E2 -1083.389} C_VEL
LIN {X 0,Y 594.366,Z 288.941,A -85,B 0,C 180,E1 -1085.428,E2 -1085.428} C_VEL
LIN {X 0,Y 594.362,Z 288.944,A -85,B 0,C 180,E1 -1087.473,E2 -1087.473} C_VEL
LIN {X 0,Y 594.331,Z 288.944,A -85,B 0,C 180,E1 -1090.217,E2 -1090.217} C_VEL
LIN {X 0,Y 594.341,Z 288.943,A -85,B 0,C 180,E1 -1092.289,E2 -1092.289} C_VEL
LIN {X 0,Y 594.34,Z 288.942,A -85,B 0,C 180,E1 -1094.378,E2 -1094.378} C_VEL
LIN {X 0,Y 594.327,Z 288.945,A -85,B 0,C 180,E1 -1097.195,E2 -1097.195} C_VEL
LIN {X 0,Y 594.359,Z 288.951,A -85,B 0,C 180,E1 -1100.054,E2 -1100.054} C_VEL
LIN {X 0,Y 594.347,Z 288.944,A -85,B 0,C 180,E1 -1102.968,E2 -1102.968} C_VEL
LIN {X 0,Y 594.319,Z 288.947,A -85,B 0,C 180,E1 -1105.195,E2 -1105.195} C_VEL
LIN {X 0,Y 594.343,Z 288.944,A -85,B 0,C 180,E1 -1107.518,E2 -1107.518} C_VEL
LIN {X 0,Y 594.331,Z 288.944,A -85,B 0,C 180,E1 -1109.779,E2 -1109.779} C_VEL
LIN {X 0,Y 594.34,Z 288.942,A -85,B 0,C 180,E1 -1112.148,E2 -1112.148} C_VEL
LIN {X 0,Y 594.359,Z 288.941,A -85,B 0,C 180,E1 -1114.581,E2 -1114.581} C_VEL
LIN {X 0,Y 594.377,Z 288.949,A -85,B 0,C 180,E1 -1117.606,E2 -1117.606} C_VEL
LIN {X 0,Y 594.349,Z 288.944,A -85,B 0,C 180,E1 -1120.568,E2 -1120.568} C_VEL
LIN {X 0,Y 594.319,Z 288.946,A -85,B 0,C 180,E1 -1122.847,E2 -1122.847} C_VEL
LIN {X 0,Y 594.314,Z 288.946,A -85,B 0,C 180,E1 -1125.196,E2 -1125.196} C_VEL
LIN {X 0,Y 594.366,Z 288.944,A -85,B 0,C 180,E1 -1128.153,E2 -1128.153} C_VEL
LIN {X 0,Y 594.352,Z 288.946,A -85,B 0,C 180,E1 -1131.299,E2 -1131.299} C_VEL
LIN {X 0,Y 594.322,Z 288.947,A -85,B 0,C 180,E1 -1133.753,E2 -1133.753} C_VEL
LIN {X 0,Y 594.346,Z 288.942,A -85,B 0,C 180,E1 -1136.236,E2 -1136.236} C_VEL
LIN {X 0,Y 594.338,Z 288.944,A -85,B 0,C 180,E1 -1138.648,E2 -1138.648} C_VEL
LIN {X 0,Y 594.373,Z 288.94,A -85,B 0,C 180,E1 -1141.043,E2 -1141.043} C_VEL
LIN {X 0,Y 594.354,Z 288.954,A -85,B 0,C 180,E1 -1144.055,E2 -1144.055} C_VEL
LIN {X 0,Y 594.366,Z 288.952,A -85,B 0,C 180,E1 -1146.295,E2 -1146.295} C_VEL
LIN {X 0,Y 594.399,Z 289.135,A -85,B 0,C 180,E1 -1148.088,E2 -1148.088} C_VEL
LIN {X 0,Y 594.691,Z 292.839,A -85,B 0,C 180,E1 -1148.678,E2 -1148.678} C_VEL
LIN {X 0,Y 594.557,Z 312.23,A -85,B 0,C 180,E1 -1151.567,E2 -1151.567} C_VEL
LIN {X 0,Y 594.456,Z 332.742,A -85,B 0,C 180,E1 -1154.573,E2 -1154.573} C_VEL
LIN {X 0,Y 594.445,Z 347.278,A -85,B 0,C 180,E1 -1156.649,E2 -1156.649} C_VEL
LIN {X 0,Y 594.749,Z 350.711,A -85,B 0,C 180,E1 -1156.721,E2 -1156.721} C_VEL
LIN {X 0,Y 594.676,Z 453.058,A -85,B 0,C 180,E1 -1157.977,E2 -1157.977} C_VEL
LIN {X 0,Y 594.648,Z 463.044,A -85,B 0,C 180,E1 -1158.171,E2 -1158.171} C_VEL
LIN {X 0,Y 594.604,Z 474.258,A -85,B 0,C 180,E1 -1158.494,E2 -1158.494} C_VEL
LIN {X 0,Y 594.547,Z 484.954,A -85,B 0,C 180,E1 -1158.908,E2 -1158.908} C_VEL
LIN {X 0,Y 594.481,Z 495.645,A -85,B 0,C 180,E1 -1159.441,E2 -1159.441} C_VEL
LIN {X 0,Y 594.435,Z 504.136,A -85,B 0,C 180,E1 -1159.957,E2 -1159.957} C_VEL
LIN {X 0,Y 594.402,Z 513.47,A -85,B 0,C 180,E1 -1160.644,E2 -1160.644} C_VEL
LIN {X 0,Y 594.372,Z 521.292,A -85,B 0,C 180,E1 -1161.329,E2 -1161.329} C_VEL
LIN {X 0,Y 594.34,Z 529.411,A -85,B 0,C 180,E1 -1162.184,E2 -1162.184} C_VEL
LIN {X 0,Y 594.307,Z 536.176,A -85,B 0,C 180,E1 -1163.038,E2 -1163.038} C_VEL
LIN {X 0,Y 594.283,Z 541.835,A -85,B 0,C 180,E1 -1163.89,E2 -1163.89} C_VEL
LIN {X 0,Y 594.248,Z 547.325,A -85,B 0,C 180,E1 -1164.911,E2 -1164.911} C_VEL
LIN {X 0,Y 594.257,Z 551.641,A -85,B 0,C 180,E1 -1165.931,E2 -1165.931} C_VEL
LIN {X 0,Y 594.261,Z 553.934,A -85,B 0,C 180,E1 -1166.61,E2 -1166.61} C_VEL
LIN {X 0,Y 594.233,Z 557.19,A -85,B 0,C 180,E1 -1167.967,E2 -1167.967} C_VEL
LIN {X 0,Y 594.232,Z 558.713,A -85,B 0,C 180,E1 -1169.322,E2 -1169.322} C_VEL
LIN {X 0,Y 594.23,Z 559,A -85,B 0,C 180,E1 -1170,E2 -1170} C_VEL
LIN {X 0,Y 594.236,Z 558.136,A -85,B 0,C 180,E1 -1171.355,E2 -1171.355} C_VEL
LIN {X 0,Y 594.234,Z 557.191,A -85,B 0,C 180,E1 -1172.033,E2 -1172.033} C_VEL
LIN {X 0,Y 594.261,Z 553.935,A -85,B 0,C 180,E1 -1173.39,E2 -1173.39} C_VEL
LIN {X 0,Y 594.268,Z 550.358,A -85,B 0,C 180,E1 -1174.409,E2 -1174.409} C_VEL
LIN {X 0,Y 594.283,Z 545.665,A -85,B 0,C 180,E1 -1175.429,E2 -1175.429} C_VEL
LIN {X 0,Y 594.283,Z 540.115,A -85,B 0,C 180,E1 -1176.391,E2 -1176.391} C_VEL
LIN {X 0,Y 594.327,Z 533.675,A -85,B 0,C 180,E1 -1177.303,E2 -1177.303} C_VEL
LIN {X 0,Y 594.358,Z 526.392,A -85,B 0,C 180,E1 -1178.157,E2 -1178.157} C_VEL
LIN {X 0,Y 594.409,Z 517.529,A -85,B 0,C 180,E1 -1179.013,E2 -1179.013} C_VEL
LIN {X 0,Y 594.451,Z 509.018,A -85,B 0,C 180,E1 -1179.699,E2 -1179.699} C_VEL
LIN {X 0,Y 594.457,Z 500.107,A -85,B 0,C 180,E1 -1180.301,E2 -1180.301} C_VEL
LIN {X 0,Y 594.548,Z 490.892,A -85,B 0,C 180,E1 -1180.816,E2 -1180.816} C_VEL
LIN {X 0,Y 594.596,Z 478.975,A -85,B 0,C 180,E1 -1181.337,E2 -1181.337} C_VEL
LIN {X 0,Y 594.636,Z 468.027,A -85,B 0,C 180,E1 -1181.699,E2 -1181.699} C_VEL
LIN {X 0,Y 594.678,Z 456.962,A -85,B 0,C 180,E1 -1181.958,E2 -1181.958} C_VEL
LIN {X 0,Y 594.684,Z 440.158,A -85,B 0,C 180,E1 -1182.195,E2 -1182.195} C_VEL
LIN {X 0,Y 594.569,Z 348.194,A -85,B 0,C 180,E1 -1183.315,E2 -1183.315} C_VEL
LIN {X 0,Y 594.438,Z 347.004,A -85,B 0,C 180,E1 -1183.373,E2 -1183.373} C_VEL
LIN {X 0,Y 594.485,Z 326.71,A -85,B 0,C 180,E1 -1186.306,E2 -1186.306} C_VEL
LIN {X 0,Y 594.546,Z 309.34,A -85,B 0,C 180,E1 -1188.862,E2 -1188.862} C_VEL
LIN {X 0,Y 594.699,Z 291.718,A -85,B 0,C 180,E1 -1191.491,E2 -1191.491} C_VEL
LIN {X 0,Y 594.382,Z 289.025,A -85,B 0,C 180,E1 -1191.959,E2 -1191.959} C_VEL
LIN {X 0,Y 594.386,Z 288.941,A -85,B 0,C 180,E1 -1194.446,E2 -1194.446} C_VEL
LIN {X 0,Y 594.345,Z 288.944,A -85,B 0,C 180,E1 -1196.701,E2 -1196.701} C_VEL
LIN {X 0,Y 594.371,Z 288.94,A -85,B 0,C 180,E1 -1198.999,E2 -1198.999} C_VEL
LIN {X 0,Y 594.366,Z 288.941,A -85,B 0,C 180,E1 -1201.641,E2 -1201.641} C_VEL
LIN {X 0,Y 594.374,Z 288.952,A -85,B 0,C 180,E1 -1204.58,E2 -1204.58} C_VEL
LIN {X 0,Y 594.383,Z 288.938,A -85,B 0,C 180,E1 -1207.608,E2 -1207.608} C_VEL
LIN {X 0,Y 594.359,Z 288.945,A -85,B 0,C 180,E1 -1210.568,E2 -1210.568} C_VEL
LIN {X 0,Y 594.371,Z 288.95,A -85,B 0,C 180,E1 -1213.299,E2 -1213.299} C_VEL
LIN {X 0,Y 594.365,Z 288.941,A -85,B 0,C 180,E1 -1216.161,E2 -1216.161} C_VEL
LIN {X 0,Y 594.374,Z 288.939,A -85,B 0,C 180,E1 -1218.536,E2 -1218.536} C_VEL
LIN {X 0,Y 594.379,Z 288.942,A -85,B 0,C 180,E1 -1221.296,E2 -1221.296} C_VEL
LIN {X 0,Y 594.359,Z 288.95,A -85,B 0,C 180,E1 -1223.756,E2 -1223.756} C_VEL
LIN {X 0,Y 594.379,Z 288.949,A -85,B 0,C 180,E1 -1226.239,E2 -1226.239} C_VEL
LIN {X 0,Y 594.391,Z 288.942,A -85,B 0,C 180,E1 -1228.651,E2 -1228.651} C_VEL
LIN {X 0,Y 594.385,Z 288.94,A -85,B 0,C 180,E1 -1231.042,E2 -1231.042} C_VEL
LIN {X 0,Y 594.383,Z 288.939,A -85,B 0,C 180,E1 -1233.978,E2 -1233.978} C_VEL
LIN {X 0,Y 594.379,Z 288.941,A -85,B 0,C 180,E1 -1236.296,E2 -1236.296} C_VEL
LIN {X 0,Y 594.403,Z 288.945,A -85,B 0,C 180,E1 -1239.225,E2 -1239.225} C_VEL
LIN {X 0,Y 594.357,Z 288.941,A -85,B 0,C 180,E1 -1242.095,E2 -1242.095} C_VEL
LIN {X 0,Y 594.369,Z 288.94,A -85,B 0,C 180,E1 -1244.219,E2 -1244.219} C_VEL
LIN {X 0,Y 594.371,Z 288.941,A -85,B 0,C 180,E1 -1247.017,E2 -1247.017} C_VEL
LIN {X 0,Y 594.392,Z 288.949,A -85,B 0,C 180,E1 -1249.784,E2 -1249.784} C_VEL
LIN {X 0,Y 594.398,Z 288.939,A -85,B 0,C 180,E1 -1252.527,E2 -1252.527} C_VEL
LIN {X 0,Y 594.398,Z 288.936,A -85,B 0,C 180,E1 -1255.253,E2 -1255.253} C_VEL
LIN {X 0,Y 594.398,Z 288.94,A -85,B 0,C 180,E1 -1257.967,E2 -1257.967} C_VEL
LIN {X 0,Y 594.424,Z 288.944,A -85,B 0,C 180,E1 -1260.678,E2 -1260.678} C_VEL
LIN {X 0,Y 594.374,Z 288.941,A -85,B 0,C 180,E1 -1263.39,E2 -1263.39} C_VEL
LIN {X 0,Y 594.392,Z 288.937,A -85,B 0,C 180,E1 -1266.109,E2 -1266.109} C_VEL
LIN {X 0,Y 594.404,Z 288.94,A -85,B 0,C 180,E1 -1268.842,E2 -1268.842} C_VEL
LIN {X 0,Y 594.395,Z 288.945,A -85,B 0,C 180,E1 -1271.596,E2 -1271.596} C_VEL
LIN {X 0,Y 594.387,Z 288.938,A -85,B 0,C 180,E1 -1274.377,E2 -1274.377} C_VEL
LIN {X 0,Y 594.36,Z 288.945,A -85,B 0,C 180,E1 -1275.33,E2 -1275.33} C_VEL
LIN {X 0,Y 593.689,Z 289.036,A -85,B 0,C 180,E1 -1275.896,E2 -1275.896} C_VEL
LIN {X 0,Y 590.835,Z 289.394,A -85,B 0,C 180,E1 -1276.814,E2 -1276.814} C_VEL
LIN {X 0,Y 588.43,Z 289.692,A -85,B 0,C 180,E1 -1277.553,E2 -1277.553} C_VEL
LIN {X 0,Y 587.402,Z 289.815,A -85,B 0,C 180,E1 -1278.123,E2 -1278.123} C_VEL
LIN {X 0,Y 587.32,Z 289.822,A -85,B 0,C 180,E1 -1278.316,E2 -1278.316} C_VEL
LIN {X 0,Y 587.333,Z 289.816,A -85,B 0,C 180,E1 -1281.038,E2 -1281.038} C_VEL
LIN {X 0,Y 587.316,Z 289.819,A -85,B 0,C 180,E1 -1283.259,E2 -1283.259} C_VEL
LIN {X 0,Y 587.337,Z 289.816,A -85,B 0,C 180,E1 -1285.517,E2 -1285.517} C_VEL
LIN {X 0,Y 587.323,Z 289.828,A -85,B 0,C 180,E1 -1288.597,E2 -1288.597} C_VEL
LIN {X 0,Y 587.327,Z 289.826,A -85,B 0,C 180,E1 -1290.967,E2 -1290.967} C_VEL
LIN {X 0,Y 587.328,Z 289.821,A -85,B 0,C 180,E1 -1293.397,E2 -1293.397} C_VEL
LIN {X 0,Y 587.288,Z 289.823,A -85,B 0,C 180,E1 -1295.9,E2 -1295.9} C_VEL
LIN {X 0,Y 587.319,Z 289.818,A -85,B 0,C 180,E1 -1298.48,E2 -1298.48} C_VEL
LIN {X 0,Y 587.336,Z 289.822,A -85,B 0,C 180,E1 -1301.157,E2 -1301.157} C_VEL
LIN {X 0,Y 587.321,Z 289.827,A -85,B 0,C 180,E1 -1304.113,E2 -1304.113} C_VEL
LIN {X 0,Y 587.364,Z 289.985,A -85,B 0,C 180,E1 -1305.56,E2 -1305.56} C_VEL
LIN {X 0,Y 587.61,Z 294.223,A -85,B 0,C 180,E1 -1306.29,E2 -1306.29} C_VEL
LIN {X 0,Y 587.486,Z 311.515,A -85,B 0,C 180,E1 -1309.121,E2 -1309.121} C_VEL
LIN {X 0,Y 587.404,Z 328.56,A -85,B 0,C 180,E1 -1311.873,E2 -1311.873} C_VEL
LIN {X 0,Y 587.384,Z 332.888,A -85,B 0,C 180,E1 -1312.533,E2 -1312.533} C_VEL
LIN {X 0,Y 587.838,Z 336.13,A -85,B 0,C 180,E1 -1312.612,E2 -1312.612} C_VEL
LIN {X 0,Y 587.742,Z 438.169,A -85,B 0,C 180,E1 -1313.88,E2 -1313.88} C_VEL
LIN {X 0,Y 587.692,Z 448.577,A -85,B 0,C 180,E1 -1314.089,E2 -1314.089} C_VEL
LIN {X 0,Y 587.653,Z 458.231,A -85,B 0,C 180,E1 -1314.364,E2 -1314.364} C_VEL
LIN {X 0,Y 587.594,Z 469.104,A -85,B 0,C 180,E1 -1314.781,E2 -1314.781} C_VEL
LIN {X 0,Y 587.495,Z 480.14,A -85,B 0,C 180,E1 -1315.33,E2 -1315.33} C_VEL
LIN {X 0,Y 587.439,Z 489.242,A -85,B 0,C 180,E1 -1315.889,E2 -1315.889} C_VEL
LIN {X 0,Y 587.398,Z 498.836,A -85,B 0,C 180,E1 -1316.607,E2 -1316.607} C_VEL
LIN {X 0,Y 587.364,Z 506.024,A -85,B 0,C 180,E1 -1317.243,E2 -1317.243} C_VEL
LIN {X 0,Y 587.285,Z 513.52,A -85,B 0,C 180,E1 -1318.026,E2 -1318.026} C_VEL
LIN {X 0,Y 587.242,Z 521.379,A -85,B 0,C 180,E1 -1319.028,E2 -1319.028} C_VEL
LIN {X 0,Y 587.212,Z 527.724,A -85,B 0,C 180,E1 -1320.021,E2 -1320.021} C_VEL
LIN {X 0,Y 587.174,Z 532.337,A -85,B 0,C 180,E1 -1320.898,E2 -1320.898} C_VEL
LIN {X 0,Y 587.184,Z 536.166,A -85,B 0,C 180,E1 -1321.785,E2 -1321.785} C_VEL
LIN {X 0,Y 587.129,Z 539.87,A -85,B 0,C 180,E1 -1322.944,E2 -1322.944} C_VEL
LIN {X 0,Y 587.121,Z 541.999,A -85,B 0,C 180,E1 -1323.867,E2 -1323.867} C_VEL
LIN {X 0,Y 587.103,Z 543.654,A -85,B 0,C 180,E1 -1325.23,E2 -1325.23} C_VEL
LIN {X 0,Y 587.112,Z 543.992,A -85,B 0,C 180,E1 -1325.984,E2 -1325.984} C_VEL
LIN {X 0,Y 587.127,Z 543.458,A -85,B 0,C 180,E1 -1327.176,E2 -1327.176} C_VEL
LIN {X 0,Y 587.145,Z 542.006,A -85,B 0,C 180,E1 -1328.219,E2 -1328.219} C_VEL
LIN {X 0,Y 587.146,Z 540.19,A -85,B 0,C 180,E1 -1329.01,E2 -1329.01} C_VEL
LIN {X 0,Y 587.163,Z 535.736,A -85,B 0,C 180,E1 -1330.419,E2 -1330.419} C_VEL
LIN {X 0,Y 587.206,Z 529.835,A -85,B 0,C 180,E1 -1331.689,E2 -1331.689} C_VEL
LIN {X 0,Y 587.243,Z 524.586,A -85,B 0,C 180,E1 -1332.591,E2 -1332.591} C_VEL
LIN {X 0,Y 587.253,Z 518.259,A -85,B 0,C 180,E1 -1333.487,E2 -1333.487} C_VEL
LIN {X 0,Y 587.288,Z 510.617,A -85,B 0,C 180,E1 -1334.38,E2 -1334.38} C_VEL
LIN {X 0,Y 587.378,Z 502.355,A -85,B 0,C 180,E1 -1335.182,E2 -1335.182} C_VEL
LIN {X 0,Y 587.419,Z 494.239,A -85,B 0,C 180,E1 -1335.846,E2 -1335.846} C_VEL
LIN {X 0,Y 587.489,Z 484.411,A -85,B 0,C 180,E1 -1336.51,E2 -1336.51} C_VEL
LIN {X 0,Y 587.561,Z 474.857,A -85,B 0,C 180,E1 -1337.04,E2 -1337.04} C_VEL
LIN {X 0,Y 587.634,Z 463.811,A -85,B 0,C 180,E1 -1337.524,E2 -1337.524} C_VEL
LIN {X 0,Y 587.725,Z 453.274,A -85,B 0,C 180,E1 -1337.877,E2 -1337.877} C_VEL
LIN {X 0,Y 587.725,Z 442.345,A -85,B 0,C 180,E1 -1338.14,E2 -1338.14} C_VEL
LIN {X 0,Y 587.775,Z 424.572,A -85,B 0,C 180,E1 -1338.393,E2 -1338.393} C_VEL
LIN {X 0,Y 587.73,Z 335.092,A -85,B 0,C 180,E1 -1339.493,E2 -1339.493} C_VEL
LIN {X 0,Y 587.403,Z 332.929,A -85,B 0,C 180,E1 -1339.552,E2 -1339.552} C_VEL
LIN {X 0,Y 587.413,Z 318.002,A -85,B 0,C 180,E1 -1341.919,E2 -1341.919} C_VEL
LIN {X 0,Y 587.506,Z 302.085,A -85,B 0,C 180,E1 -1344.508,E2 -1344.508} C_VEL
LIN {X 0,Y 587.509,Z 290.623,A -85,B 0,C 180,E1 -1346.399,E2 -1346.399} C_VEL
LIN {X 0,Y 587.369,Z 289.89,A -85,B 0,C 180,E1 -1346.57,E2 -1346.57} C_VEL
LIN {X 0,Y 587.386,Z 289.81,A -85,B 0,C 180,E1 -1349.315,E2 -1349.315} C_VEL
LIN {X 0,Y 587.365,Z 289.814,A -85,B 0,C 180,E1 -1352.057,E2 -1352.057} C_VEL
LIN {X 0,Y 587.368,Z 289.821,A -85,B 0,C 180,E1 -1354.805,E2 -1354.805} C_VEL
LIN {X 0,Y 587.366,Z 289.817,A -85,B 0,C 180,E1 -1357.563,E2 -1357.563} C_VEL
LIN {X 0,Y 587.343,Z 289.815,A -85,B 0,C 180,E1 -1360.34,E2 -1360.34} C_VEL
LIN {X 0,Y 587.317,Z 289.82,A -85,B 0,C 180,E1 -1363.142,E2 -1363.142} C_VEL
LIN {X 0,Y 587.326,Z 289.829,A -85,B 0,C 180,E1 -1365.975,E2 -1365.975} C_VEL
LIN {X 0,Y 587.351,Z 289.815,A -85,B 0,C 180,E1 -1368.849,E2 -1368.849} C_VEL
LIN {X 0,Y 587.321,Z 289.819,A -85,B 0,C 180,E1 -1371.774,E2 -1371.774} C_VEL
LIN {X 0,Y 587.35,Z 289.826,A -85,B 0,C 180,E1 -1374.759,E2 -1374.759} C_VEL
LIN {X 0,Y 587.349,Z 289.813,A -85,B 0,C 180,E1 -1377.818,E2 -1377.818} C_VEL
LIN {X 0,Y 587.33,Z 289.817,A -85,B 0,C 180,E1 -1380.509,E2 -1380.509} C_VEL
LIN {X 0,Y 587.339,Z 289.821,A -85,B 0,C 180,E1 -1383.112,E2 -1383.112} C_VEL
LIN {X 0,Y 587.299,Z 289.83,A -85,B 0,C 180,E1 -1385.538,E2 -1385.538} C_VEL
LIN {X 0,Y 587.323,Z 289.819,A -85,B 0,C 180,E1 -1388.48,E2 -1388.48} C_VEL
LIN {X 0,Y 587.333,Z 289.814,A -85,B 0,C 180,E1 -1391.157,E2 -1391.157} C_VEL
LIN {X 0,Y 587.32,Z 289.824,A -85,B 0,C 180,E1 -1394.113,E2 -1394.113} C_VEL
LIN {X 0,Y 587.301,Z 289.825,A -85,B 0,C 180,E1 -1396.992,E2 -1396.992} C_VEL
LIN {X 0,Y 587.31,Z 289.817,A -85,B 0,C 180,E1 -1399.745,E2 -1399.745} C_VEL
LIN {X 0,Y 587.342,Z 289.815,A -85,B 0,C 180,E1 -1402.392,E2 -1402.392} C_VEL
LIN {X 0,Y 587.34,Z 289.822,A -85,B 0,C 180,E1 -1405.654,E2 -1405.654} C_VEL
LIN {X 0,Y 587.341,Z 289.816,A -85,B 0,C 180,E1 -1408.231,E2 -1408.231} C_VEL
LIN {X 0,Y 587.347,Z 289.811,A -85,B 0,C 180,E1 -1410.868,E2 -1410.868} C_VEL
LIN {X 0,Y 587.316,Z 289.824,A -85,B 0,C 180,E1 -1413.828,E2 -1413.828} C_VEL
LIN {X 0,Y 587.331,Z 289.822,A -85,B 0,C 180,E1 -1415.993,E2 -1415.993} C_VEL
LIN {X 0,Y 587.334,Z 289.819,A -85,B 0,C 180,E1 -1418.962,E2 -1418.962} C_VEL
LIN {X 0,Y 587.339,Z 289.817,A -85,B 0,C 180,E1 -1421.151,E2 -1421.151} C_VEL
LIN {X 0,Y 587.306,Z 289.818,A -85,B 0,C 180,E1 -1424.024,E2 -1424.024} C_VEL
LIN {X 0,Y 587.339,Z 289.815,A -85,B 0,C 180,E1 -1426.154,E2 -1426.154} C_VEL
LIN {X 0,Y 587.349,Z 289.817,A -85,B 0,C 180,E1 -1428.962,E2 -1428.962} C_VEL
LIN {X 0,Y 587.328,Z 289.826,A -85,B 0,C 180,E1 -1431.744,E2 -1431.744} C_VEL
LIN {X 0,Y 587.333,Z 289.816,A -85,B 0,C 180,E1 -1434.507,E2 -1434.507} C_VEL
LIN {X 0,Y 587.347,Z 289.814,A -85,B 0,C 180,E1 -1437.256,E2 -1437.256} C_VEL
LIN {X 0,Y 587.382,Z 289.814,A -85,B 0,C 180,E1 -1440,E2 -1440} C_VEL
LIN {X 0,Y 587.369,Z 289.82,A -85,B 0,C 180,E1 -1442.743,E2 -1442.743} C_VEL
LIN {X 0,Y 587.332,Z 289.816,A -85,B 0,C 180,E1 -1445.493,E2 -1445.493} C_VEL
LIN {X 0,Y 587.317,Z 289.821,A -85,B 0,C 180,E1 -1447.564,E2 -1447.564} C_VEL
LIN {X 0,Y 587.293,Z 289.821,A -85,B 0,C 180,E1 -1450.341,E2 -1450.341} C_VEL
LIN {X 0,Y 587.297,Z 289.82,A -85,B 0,C 180,E1 -1452.439,E2 -1452.439} C_VEL
LIN {X 0,Y 587.308,Z 289.817,A -85,B 0,C 180,E1 -1454.554,E2 -1454.554} C_VEL
LIN {X 0,Y 587.278,Z 289.825,A -85,B 0,C 180,E1 -1457.408,E2 -1457.408} C_VEL
LIN {X 0,Y 587.301,Z 289.823,A -85,B 0,C 180,E1 -1459.576,E2 -1459.576} C_VEL
LIN {X 0,Y 587.333,Z 289.824,A -85,B 0,C 180,E1 -1462.514,E2 -1462.514} C_VEL
LIN {X 0,Y 587.306,Z 289.827,A -85,B 0,C 180,E1 -1464.76,E2 -1464.76} C_VEL
LIN {X 0,Y 587.298,Z 289.821,A -85,B 0,C 180,E1 -1467.682,E2 -1467.682} C_VEL
LIN {X 0,Y 587.292,Z 289.82,A -85,B 0,C 180,E1 -1470.172,E2 -1470.172} C_VEL
LIN {X 0,Y 587.331,Z 289.824,A -85,B 0,C 180,E1 -1473.11,E2 -1473.11} C_VEL
LIN {X 0,Y 587.274,Z 289.828,A -85,B 0,C 180,E1 -1475.901,E2 -1475.901} C_VEL
LIN {X 0,Y 587.3,Z 289.821,A -85,B 0,C 180,E1 -1478.481,E2 -1478.481} C_VEL
LIN {X 0,Y 587.304,Z 289.82,A -85,B 0,C 180,E1 -1481.159,E2 -1481.159} C_VEL
LIN {X 0,Y 587.301,Z 289.829,A -85,B 0,C 180,E1 -1484.111,E2 -1484.111} C_VEL
LIN {X 0,Y 587.272,Z 289.827,A -85,B 0,C 180,E1 -1486.99,E2 -1486.99} C_VEL
LIN {X 0,Y 587.291,Z 289.821,A -85,B 0,C 180,E1 -1489.744,E2 -1489.744} C_VEL
LIN {X 0,Y 587.33,Z 289.818,A -85,B 0,C 180,E1 -1492.391,E2 -1492.391} C_VEL
LIN {X 0,Y 587.324,Z 289.82,A -85,B 0,C 180,E1 -1495.777,E2 -1495.777} C_VEL
LIN {X 0,Y 587.329,Z 289.818,A -85,B 0,C 180,E1 -1498.23,E2 -1498.23} C_VEL
LIN {X 0,Y 587.338,Z 289.816,A -85,B 0,C 180,E1 -1500.868,E2 -1500.868} C_VEL
LIN {X 0,Y 587.308,Z 289.829,A -85,B 0,C 180,E1 -1503.829,E2 -1503.829} C_VEL
LIN {X 0,Y 587.314,Z 289.829,A -85,B 0,C 180,E1 -1505.992,E2 -1505.992} C_VEL
LIN {X 0,Y 587.358,Z 290.028,A -85,B 0,C 180,E1 -1507.95,E2 -1507.95} C_VEL
LIN {X 0,Y 587.747,Z 294.35,A -85,B 0,C 180,E1 -1508.644,E2 -1508.644} C_VEL
LIN {X 0,Y 587.567,Z 311.023,A -85,B 0,C 180,E1 -1511.158,E2 -1511.158} C_VEL
LIN {X 0,Y 587.483,Z 329.122,A -85,B 0,C 180,E1 -1513.851,E2 -1513.851} C_VEL
LIN {X 0,Y 587.395,Z 347.272,A -85,B 0,C 180,E1 -1516.486,E2 -1516.486} C_VEL
LIN {X 0,Y 587.837,Z 350.711,A -85,B 0,C 180,E1 -1516.562,E2 -1516.562} C_VEL
LIN {X 0,Y 587.754,Z 453.058,A -85,B 0,C 180,E1 -1517.834,E2 -1517.834} C_VEL
LIN {X 0,Y 587.716,Z 463.043,A -85,B 0,C 180,E1 -1518.03,E2 -1518.03} C_VEL
LIN {X 0,Y 587.664,Z 473.14,A -85,B 0,C 180,E1 -1518.315,E2 -1518.315} C_VEL
LIN {X 0,Y 587.574,Z 484.51,A -85,B 0,C 180,E1 -1518.754,E2 -1518.754} C_VEL
LIN {X 0,Y 587.522,Z 494.143,A -85,B 0,C 180,E1 -1519.228,E2 -1519.228} C_VEL
LIN {X 0,Y 587.412,Z 504.132,A -85,B 0,C 180,E1 -1519.835,E2 -1519.835} C_VEL
LIN {X 0,Y 587.378,Z 513.467,A -85,B 0,C 180,E1 -1520.531,E2 -1520.531} C_VEL
LIN {X 0,Y 587.33,Z 521.291,A -85,B 0,C 180,E1 -1521.224,E2 -1521.224} C_VEL
LIN {X 0,Y 587.283,Z 529.412,A -85,B 0,C 180,E1 -1522.09,E2 -1522.09} C_VEL
LIN {X 0,Y 587.242,Z 536.177,A -85,B 0,C 180,E1 -1522.954,E2 -1522.954} C_VEL
LIN {X 0,Y 587.213,Z 541.836,A -85,B 0,C 180,E1 -1523.816,E2 -1523.816} C_VEL
LIN {X 0,Y 587.161,Z 547.325,A -85,B 0,C 180,E1 -1524.849,E2 -1524.849} C_VEL
LIN {X 0,Y 587.177,Z 551.641,A -85,B 0,C 180,E1 -1525.882,E2 -1525.882} C_VEL
LIN {X 0,Y 587.187,Z 553.935,A -85,B 0,C 180,E1 -1526.569,E2 -1526.569} C_VEL
LIN {X 0,Y 587.133,Z 557.189,A -85,B 0,C 180,E1 -1527.942,E2 -1527.942} C_VEL
LIN {X 0,Y 587.133,Z 558.713,A -85,B 0,C 180,E1 -1529.314,E2 -1529.314} C_VEL
LIN {X 0,Y 587.131,Z 559,A -85,B 0,C 180,E1 -1530,E2 -1530} C_VEL
LIN {X 0,Y 587.136,Z 558.137,A -85,B 0,C 180,E1 -1531.372,E2 -1531.372} C_VEL
LIN {X 0,Y 587.133,Z 557.19,A -85,B 0,C 180,E1 -1532.058,E2 -1532.058} C_VEL
LIN {X 0,Y 587.187,Z 553.936,A -85,B 0,C 180,E1 -1533.431,E2 -1533.431} C_VEL
LIN {X 0,Y 587.186,Z 550.358,A -85,B 0,C 180,E1 -1534.462,E2 -1534.462} C_VEL
LIN {X 0,Y 587.205,Z 545.665,A -85,B 0,C 180,E1 -1535.494,E2 -1535.494} C_VEL
LIN {X 0,Y 587.242,Z 539.044,A -85,B 0,C 180,E1 -1536.626,E2 -1536.626} C_VEL
LIN {X 0,Y 587.26,Z 533.674,A -85,B 0,C 180,E1 -1537.392,E2 -1537.392} C_VEL
LIN {X 0,Y 587.292,Z 526.392,A -85,B 0,C 180,E1 -1538.256,E2 -1538.256} C_VEL
LIN {X 0,Y 587.372,Z 517.531,A -85,B 0,C 180,E1 -1539.122,E2 -1539.122} C_VEL
LIN {X 0,Y 587.436,Z 509.022,A -85,B 0,C 180,E1 -1539.816,E2 -1539.816} C_VEL
LIN {X 0,Y 587.473,Z 500.111,A -85,B 0,C 180,E1 -1540.425,E2 -1540.425} C_VEL
LIN {X 0,Y 587.571,Z 490.897,A -85,B 0,C 180,E1 -1540.946,E2 -1540.946} C_VEL
LIN {X 0,Y 587.628,Z 479.485,A -85,B 0,C 180,E1 -1541.455,E2 -1541.455} C_VEL
LIN {X 0,Y 587.683,Z 468.028,A -85,B 0,C 180,E1 -1541.839,E2 -1541.839} C_VEL
LIN {X 0,Y 587.758,Z 456.96,A -85,B 0,C 180,E1 -1542.1,E2 -1542.1} C_VEL
LIN {X 0,Y 587.746,Z 440.158,A -85,B 0,C 180,E1 -1542.342,E2 -1542.342} C_VEL
LIN {X 0,Y 587.691,Z 349.156,A -85,B 0,C 180,E1 -1543.46,E2 -1543.46} C_VEL
LIN {X 0,Y 587.395,Z 347.269,A -85,B 0,C 180,E1 -1543.514,E2 -1543.514} C_VEL
LIN {X 0,Y 587.483,Z 329.123,A -85,B 0,C 180,E1 -1546.149,E2 -1546.149} C_VEL
LIN {X 0,Y 587.566,Z 311.024,A -85,B 0,C 180,E1 -1548.842,E2 -1548.842} C_VEL
LIN {X 0,Y 587.76,Z 294.118,A -85,B 0,C 180,E1 -1551.391,E2 -1551.391} C_VEL
LIN {X 0,Y 587.363,Z 289.951,A -85,B 0,C 180,E1 -1552.073,E2 -1552.073} C_VEL
LIN {X 0,Y 587.305,Z 289.822,A -85,B 0,C 180,E1 -1554.761,E2 -1554.761} C_VEL
LIN {X 0,Y 587.298,Z 289.827,A -85,B 0,C 180,E1 -1557.684,E2 -1557.684} C_VEL
LIN {X 0,Y 587.312,Z 289.831,A -85,B 0,C 180,E1 -1560.171,E2 -1560.171} C_VEL
LIN {X 0,Y 587.337,Z 289.825,A -85,B 0,C 180,E1 -1562.579,E2 -1562.579} C_VEL
LIN {X 0,Y 587.321,Z 289.822,A -85,B 0,C 180,E1 -1565.056,E2 -1565.056} C_VEL
LIN {X 0,Y 587.328,Z 289.817,A -85,B 0,C 180,E1 -1567.837,E2 -1567.837} C_VEL
LIN {X 0,Y 587.308,Z 289.82,A -85,B 0,C 180,E1 -1570.255,E2 -1570.255} C_VEL
LIN {X 0,Y 587.31,Z 289.831,A -85,B 0,C 180,E1 -1573.118,E2 -1573.118} C_VEL
LIN {X 0,Y 587.321,Z 289.819,A -85,B 0,C 180,E1 -1576.05,E2 -1576.05} C_VEL
LIN {X 0,Y 587.331,Z 289.818,A -85,B 0,C 180,E1 -1578.926,E2 -1578.926} C_VEL
LIN {X 0,Y 587.327,Z 289.824,A -85,B 0,C 180,E1 -1581.521,E2 -1581.521} C_VEL
LIN {X 0,Y 587.298,Z 289.83,A -85,B 0,C 180,E1 -1584.101,E2 -1584.101} C_VEL
LIN {X 0,Y 587.334,Z 289.82,A -85,B 0,C 180,E1 -1586.604,E2 -1586.604} C_VEL
LIN {X 0,Y 587.342,Z 289.815,A -85,B 0,C 180,E1 -1589.489,E2 -1589.489} C_VEL
LIN {X 0,Y 587.352,Z 289.821,A -85,B 0,C 180,E1 -1592.307,E2 -1592.307} C_VEL
LIN {X 0,Y 587.352,Z 289.817,A -85,B 0,C 180,E1 -1595.242,E2 -1595.242} C_VEL
LIN {X 0,Y 587.323,Z 289.818,A -85,B 0,C 180,E1 -1598.226,E2 -1598.226} C_VEL
LIN {X 0,Y 587.351,Z 289.826,A -85,B 0,C 180,E1 -1601.151,E2 -1601.151} C_VEL
LIN {X 0,Y 587.326,Z 289.819,A -85,B 0,C 180,E1 -1604.025,E2 -1604.025} C_VEL
LIN {X 0,Y 587.363,Z 289.814,A -85,B 0,C 180,E1 -1606.155,E2 -1606.155} C_VEL
LIN {X 0,Y 587.344,Z 289.815,A -85,B 0,C 180,E1 -1608.963,E2 -1608.963} C_VEL
LIN {X 0,Y 587.374,Z 289.818,A -85,B 0,C 180,E1 -1611.745,E2 -1611.745} C_VEL
LIN {X 0,Y 587.358,Z 289.818,A -85,B 0,C 180,E1 -1614.507,E2 -1614.507} C_VEL
LIN {X 0,Y 587.378,Z 289.811,A -85,B 0,C 180,E1 -1617.257,E2 -1617.257} C_VEL
LIN {X 0,Y 587.388,Z 289.812,A -85,B 0,C 180,E1 -1620,E2 -1620} C_VEL
LIN {X 0,Y 587.377,Z 289.823,A -85,B 0,C 180,E1 -1622.743,E2 -1622.743} C_VEL
LIN {X 0,Y 587.36,Z 289.816,A -85,B 0,C 180,E1 -1625.493,E2 -1625.493} C_VEL
LIN {X 0,Y 587.371,Z 289.811,A -85,B 0,C 180,E1 -1628.255,E2 -1628.255} C_VEL
LIN {X 0,Y 587.351,Z 289.822,A -85,B 0,C 180,E1 -1631.134,E2 -1631.134} C_VEL
LIN {X 0,Y 587.359,Z 289.815,A -85,B 0,C 180,E1 -1634.257,E2 -1634.257} C_VEL
LIN {X 0,Y 587.352,Z 289.818,A -85,B 0,C 180,E1 -1637.406,E2 -1637.406} C_VEL
LIN {X 0,Y 587.32,Z 289.822,A -85,B 0,C 180,E1 -1638.316,E2 -1638.316} C_VEL
LIN {X 0,Y 586.667,Z 289.901,A -85,B 0,C 180,E1 -1638.888,E2 -1638.888} C_VEL
LIN {X 0,Y 583.838,Z 290.26,A -85,B 0,C 180,E1 -1639.816,E2 -1639.816} C_VEL
LIN {X 0,Y 581.431,Z 290.555,A -85,B 0,C 180,E1 -1640.563,E2 -1640.563} C_VEL
LIN {X 0,Y 580.379,Z 290.683,A -85,B 0,C 180,E1 -1641.139,E2 -1641.139} C_VEL
LIN {X 0,Y 580.285,Z 290.695,A -85,B 0,C 180,E1 -1641.334,E2 -1641.334} C_VEL
LIN {X 0,Y 580.3,Z 290.705,A -85,B 0,C 180,E1 -1644.316,E2 -1644.316} C_VEL
LIN {X 0,Y 580.269,Z 290.705,A -85,B 0,C 180,E1 -1646.624,E2 -1646.624} C_VEL
LIN {X 0,Y 580.298,Z 290.695,A -85,B 0,C 180,E1 -1649.309,E2 -1649.309} C_VEL
LIN {X 0,Y 580.298,Z 290.694,A -85,B 0,C 180,E1 -1652.201,E2 -1652.201} C_VEL
LIN {X 0,Y 580.287,Z 290.699,A -85,B 0,C 180,E1 -1654.697,E2 -1654.697} C_VEL
LIN {X 0,Y 580.297,Z 290.705,A -85,B 0,C 180,E1 -1657.269,E2 -1657.269} C_VEL
LIN {X 0,Y 580.289,Z 290.695,A -85,B 0,C 180,E1 -1660.27,E2 -1660.27} C_VEL
LIN {X 0,Y 580.274,Z 290.697,A -85,B 0,C 180,E1 -1662.707,E2 -1662.707} C_VEL
LIN {X 0,Y 580.335,Z 290.9,A -85,B 0,C 180,E1 -1665.459,E2 -1665.459} C_VEL
LIN {X 0,Y 580.644,Z 295.005,A -85,B 0,C 180,E1 -1666.174,E2 -1666.174} C_VEL
LIN {X 0,Y 580.487,Z 313.104,A -85,B 0,C 180,E1 -1669.173,E2 -1669.173} C_VEL
LIN {X 0,Y 580.353,Z 332.604,A -85,B 0,C 180,E1 -1672.34,E2 -1672.34} C_VEL
LIN {X 0,Y 580.521,Z 334.091,A -85,B 0,C 180,E1 -1672.412,E2 -1672.412} C_VEL
LIN {X 0,Y 580.94,Z 338.537,A -85,B 0,C 180,E1 -1672.48,E2 -1672.48} C_VEL
LIN {X 0,Y 580.819,Z 438.254,A -85,B 0,C 180,E1 -1673.735,E2 -1673.735} C_VEL
LIN {X 0,Y 580.746,Z 448.627,A -85,B 0,C 180,E1 -1673.945,E2 -1673.945} C_VEL
LIN {X 0,Y 580.692,Z 459.084,A -85,B 0,C 180,E1 -1674.253,E2 -1674.253} C_VEL
LIN {X 0,Y 580.647,Z 469.018,A -85,B 0,C 180,E1 -1674.64,E2 -1674.64} C_VEL
LIN {X 0,Y 580.551,Z 478.611,A -85,B 0,C 180,E1 -1675.11,E2 -1675.11} C_VEL
LIN {X 0,Y 580.429,Z 488.81,A -85,B 0,C 180,E1 -1675.734,E2 -1675.734} C_VEL
LIN {X 0,Y 580.383,Z 498.289,A -85,B 0,C 180,E1 -1676.445,E2 -1676.445} C_VEL
LIN {X 0,Y 580.333,Z 506.502,A -85,B 0,C 180,E1 -1677.185,E2 -1677.185} C_VEL
LIN {X 0,Y 580.238,Z 513.938,A -85,B 0,C 180,E1 -1677.98,E2 -1677.98} C_VEL
LIN {X 0,Y 580.178,Z 520.442,A -85,B 0,C 180,E1 -1678.803,E2 -1678.803} C_VEL
LIN {X 0,Y 580.15,Z 527.02,A -85,B 0,C 180,E1 -1679.819,E2 -1679.819} C_VEL
LIN {X 0,Y 580.105,Z 531.861,A -85,B 0,C 180,E1 -1680.725,E2 -1680.725} C_VEL
LIN {X 0,Y 580.084,Z 536.398,A -85,B 0,C 180,E1 -1681.803,E2 -1681.803} C_VEL
LIN {X 0,Y 580.062,Z 538.986,A -85,B 0,C 180,E1 -1682.587,E2 -1682.587} C_VEL
LIN {X 0,Y 580.046,Z 541.74,A -85,B 0,C 180,E1 -1683.715,E2 -1683.715} C_VEL
LIN {X 0,Y 580.008,Z 543.466,A -85,B 0,C 180,E1 -1684.906,E2 -1684.906} C_VEL
LIN {X 0,Y 580.009,Z 543.857,A -85,B 0,C 180,E1 -1685.671,E2 -1685.671} C_VEL
LIN {X 0,Y 580.054,Z 543.461,A -85,B 0,C 180,E1 -1687.188,E2 -1687.188} C_VEL
LIN {X 0,Y 580.034,Z 542.451,A -85,B 0,C 180,E1 -1687.938,E2 -1687.938} C_VEL
LIN {X 0,Y 580.082,Z 539.223,A -85,B 0,C 180,E1 -1689.43,E2 -1689.43} C_VEL
LIN {X 0,Y 580.082,Z 535.46,A -85,B 0,C 180,E1 -1690.538,E2 -1690.538} C_VEL
LIN {X 0,Y 580.141,Z 530.475,A -85,B 0,C 180,E1 -1691.641,E2 -1691.641} C_VEL
LIN {X 0,Y 580.181,Z 524.149,A -85,B 0,C 180,E1 -1692.736,E2 -1692.736} C_VEL
LIN {X 0,Y 580.216,Z 517.727,A -85,B 0,C 180,E1 -1693.644,E2 -1693.644} C_VEL
LIN {X 0,Y 580.248,Z 509.997,A -85,B 0,C 180,E1 -1694.546,E2 -1694.546} C_VEL
LIN {X 0,Y 580.357,Z 502.654,A -85,B 0,C 180,E1 -1695.268,E2 -1695.268} C_VEL
LIN {X 0,Y 580.419,Z 493.96,A -85,B 0,C 180,E1 -1695.985,E2 -1695.985} C_VEL
LIN {X 0,Y 580.502,Z 484.842,A -85,B 0,C 180,E1 -1696.612,E2 -1696.612} C_VEL
LIN {X 0,Y 580.574,Z 475.402,A -85,B 0,C 180,E1 -1697.148,E2 -1697.148} C_VEL
LIN {X 0,Y 580.681,Z 464.489,A -85,B 0,C 180,E1 -1697.639,E2 -1697.639} C_VEL
LIN {X 0,Y 580.779,Z 453.375,A -85,B 0,C 180,E1 -1698.018,E2 -1698.018} C_VEL
LIN {X 0,Y 580.805,Z 442.894,A -85,B 0,C 180,E1 -1698.276,E2 -1698.276} C_VEL
LIN {X 0,Y 580.863,Z 426.498,A -85,B 0,C 180,E1 -1698.519,E2 -1698.519} C_VEL
LIN {X 0,Y 580.862,Z 336.08,A -85,B 0,C 180,E1 -1699.643,E2 -1699.643} C_VEL
LIN {X 0,Y 580.373,Z 333.059,A -85,B 0,C 180,E1 -1699.711,E2 -1699.711} C_VEL
LIN {X 0,Y 580.361,Z 328.425,A -85,B 0,C 180,E1 -1700.415,E2 -1700.415} C_VEL
LIN {X 0,Y 580.494,Z 311.965,A -85,B 0,C 180,E1 -1703.105,E2 -1703.105} C_VEL
LIN {X 0,Y 580.613,Z 294.454,A -85,B 0,C 180,E1 -1706.009,E2 -1706.009} C_VEL
LIN {X 0,Y 580.332,Z 290.81,A -85,B 0,C 180,E1 -1706.659,E2 -1706.659} C_VEL
LIN {X 0,Y 580.358,Z 290.686,A -85,B 0,C 180,E1 -1709.306,E2 -1709.306} C_VEL
LIN {X 0,Y 580.336,Z 290.69,A -85,B 0,C 180,E1 -1712.082,E2 -1712.082} C_VEL
LIN {X 0,Y 580.339,Z 290.698,A -85,B 0,C 180,E1 -1714.863,E2 -1714.863} C_VEL
LIN {X 0,Y 580.326,Z 290.693,A -85,B 0,C 180,E1 -1717.655,E2 -1717.655} C_VEL
LIN {X 0,Y 580.301,Z 290.692,A -85,B 0,C 180,E1 -1720.467,E2 -1720.467} C_VEL
LIN {X 0,Y 580.305,Z 290.691,A -85,B 0,C 180,E1 -1722.591,E2 -1722.591} C_VEL
LIN {X 0,Y 580.288,Z 290.694,A -85,B 0,C 180,E1 -1724.734,E2 -1724.734} C_VEL
LIN {X 0,Y 580.3,Z 290.696,A -85,B 0,C 180,E1 -1727.624,E2 -1727.624} C_VEL
LIN {X 0,Y 580.291,Z 290.697,A -85,B 0,C 180,E1 -1729.823,E2 -1729.823} C_VEL
LIN {X 0,Y 580.272,Z 290.7,A -85,B 0,C 180,E1 -1732.053,E2 -1732.053} C_VEL
LIN {X 0,Y 580.303,Z 290.697,A -85,B 0,C 180,E1 -1735.08,E2 -1735.08} C_VEL
LIN {X 0,Y 580.301,Z 290.691,A -85,B 0,C 180,E1 -1738.186,E2 -1738.186} C_VEL
LIN {X 0,Y 580.284,Z 290.697,A -85,B 0,C 180,E1 -1740.694,E2 -1740.694} C_VEL
LIN {X 0,Y 580.304,Z 290.701,A -85,B 0,C 180,E1 -1743.316,E2 -1743.316} C_VEL
LIN {X 0,Y 580.248,Z 290.709,A -85,B 0,C 180,E1 -1745.756,E2 -1745.756} C_VEL
LIN {X 0,Y 580.288,Z 290.7,A -85,B 0,C 180,E1 -1748.147,E2 -1748.147} C_VEL
LIN {X 0,Y 580.296,Z 290.692,A -85,B 0,C 180,E1 -1750.844,E2 -1750.844} C_VEL
LIN {X 0,Y 580.27,Z 290.696,A -85,B 0,C 180,E1 -1753.659,E2 -1753.659} C_VEL
LIN {X 0,Y 580.27,Z 290.708,A -85,B 0,C 180,E1 -1756.61,E2 -1756.61} C_VEL
LIN {X 0,Y 580.299,Z 290.696,A -85,B 0,C 180,E1 -1759.157,E2 -1759.157} C_VEL
LIN {X 0,Y 580.287,Z 290.693,A -85,B 0,C 180,E1 -1761.928,E2 -1761.928} C_VEL
LIN {X 0,Y 580.251,Z 290.698,A -85,B 0,C 180,E1 -1764.453,E2 -1764.453} C_VEL
LIN {X 0,Y 580.29,Z 290.696,A -85,B 0,C 180,E1 -1766.975,E2 -1766.975} C_VEL
LIN {X 0,Y 580.296,Z 290.697,A -85,B 0,C 180,E1 -1769.425,E2 -1769.425} C_VEL
LIN {X 0,Y 580.26,Z 290.705,A -85,B 0,C 180,E1 -1772.149,E2 -1772.149} C_VEL
LIN {X 0,Y 580.323,Z 290.689,A -85,B 0,C 180,E1 -1775.27,E2 -1775.27} C_VEL
LIN {X 0,Y 580.258,Z 290.7,A -85,B 0,C 180,E1 -1777.947,E2 -1777.947} C_VEL
LIN {X 0,Y 580.293,Z 290.698,A -85,B 0,C 180,E1 -1780.913,E2 -1780.913} C_VEL
LIN {X 0,Y 580.258,Z 290.696,A -85,B 0,C 180,E1 -1783.825,E2 -1783.825} C_VEL
LIN {X 0,Y 580.298,Z 290.692,A -85,B 0,C 180,E1 -1785.982,E2 -1785.982} C_VEL
LIN {X 0,Y 580.309,Z 290.693,A -85,B 0,C 180,E1 -1788.827,E2 -1788.827} C_VEL
LIN {X 0,Y 580.3,Z 290.703,A -85,B 0,C 180,E1 -1791.643,E2 -1791.643} C_VEL
LIN {X 0,Y 580.302,Z 290.692,A -85,B 0,C 180,E1 -1794.44,E2 -1794.44} C_VEL
LIN {X 0,Y 580.314,Z 290.689,A -85,B 0,C 180,E1 -1797.223,E2 -1797.223} C_VEL
LIN {X 0,Y 580.358,Z 290.692,A -85,B 0,C 180,E1 -1800.694,E2 -1800.694} C_VEL
LIN {X 0,Y 580.332,Z 290.695,A -85,B 0,C 180,E1 -1802.776,E2 -1802.776} C_VEL
LIN {X 0,Y 580.299,Z 290.691,A -85,B 0,C 180,E1 -1805.56,E2 -1805.56} C_VEL
LIN {X 0,Y 580.267,Z 290.698,A -85,B 0,C 180,E1 -1807.656,E2 -1807.656} C_VEL
LIN {X 0,Y 580.263,Z 290.697,A -85,B 0,C 180,E1 -1810.467,E2 -1810.467} C_VEL
LIN {X 0,Y 580.27,Z 290.695,A -85,B 0,C 180,E1 -1812.592,E2 -1812.592} C_VEL
LIN {X 0,Y 580.272,Z 290.699,A -85,B 0,C 180,E1 -1815.453,E2 -1815.453} C_VEL
LIN {X 0,Y 580.241,Z 290.705,A -85,B 0,C 180,E1 -1818.356,E2 -1818.356} C_VEL
LIN {X 0,Y 580.273,Z 290.695,A -85,B 0,C 180,E1 -1821.157,E2 -1821.157} C_VEL
LIN {X 0,Y 580.262,Z 290.695,A -85,B 0,C 180,E1 -1823.558,E2 -1823.558} C_VEL
LIN {X 0,Y 580.249,Z 290.703,A -85,B 0,C 180,E1 -1826.325,E2 -1826.325} C_VEL
LIN {X 0,Y 580.268,Z 290.701,A -85,B 0,C 180,E1 -1829.303,E2 -1829.303} C_VEL
LIN {X 0,Y 580.283,Z 290.693,A -85,B 0,C 180,E1 -1832.201,E2 -1832.201} C_VEL
LIN {X 0,Y 580.273,Z 290.696,A -85,B 0,C 180,E1 -1834.697,E2 -1834.697} C_VEL
LIN {X 0,Y 580.281,Z 290.699,A -85,B 0,C 180,E1 -1837.269,E2 -1837.269} C_VEL
LIN {X 0,Y 580.278,Z 290.7,A -85,B 0,C 180,E1 -1840.269,E2 -1840.269} C_VEL
LIN {X 0,Y 580.247,Z 290.701,A -85,B 0,C 180,E1 -1842.709,E2 -1842.709} C_VEL
LIN {X 0,Y 580.236,Z 290.701,A -85,B 0,C 180,E1 -1845.612,E2 -1845.612} C_VEL
LIN {X 0,Y 580.239,Z 290.705,A -85,B 0,C 180,E1 -1848.227,E2 -1848.227} C_VEL
LIN {X 0,Y 580.261,Z 290.708,A -85,B 0,C 180,E1 -1850.963,E2 -1850.963} C_VEL
LIN {X 0,Y 580.237,Z 290.703,A -85,B 0,C 180,E1 -1853.594,E2 -1853.594} C_VEL
LIN {X 0,Y 580.272,Z 290.695,A -85,B 0,C 180,E1 -1856.142,E2 -1856.142} C_VEL
LIN {X 0,Y 580.259,Z 290.698,A -85,B 0,C 180,E1 -1858.613,E2 -1858.613} C_VEL
LIN {X 0,Y 580.281,Z 290.696,A -85,B 0,C 180,E1 -1861.023,E2 -1861.023} C_VEL
LIN {X 0,Y 580.249,Z 290.709,A -85,B 0,C 180,E1 -1864.149,E2 -1864.149} C_VEL
LIN {X 0,Y 580.261,Z 290.708,A -85,B 0,C 180,E1 -1866.441,E2 -1866.441} C_VEL
LIN {X 0,Y 580.312,Z 290.923,A -85,B 0,C 180,E1 -1867.808,E2 -1867.808} C_VEL
LIN {X 0,Y 580.802,Z 295.459,A -85,B 0,C 180,E1 -1868.547,E2 -1868.547} C_VEL
LIN {X 0,Y 580.611,Z 312.23,A -85,B 0,C 180,E1 -1871.107,E2 -1871.107} C_VEL
LIN {X 0,Y 580.471,Z 330.329,A -85,B 0,C 180,E1 -1873.831,E2 -1873.831} C_VEL
LIN {X 0,Y 580.401,Z 347.275,A -85,B 0,C 180,E1 -1876.32,E2 -1876.32} C_VEL
LIN {X 0,Y 580.951,Z 352.5,A -85,B 0,C 180,E1 -1876.422,E2 -1876.422} C_VEL
LIN {X 0,Y 580.829,Z 453.058,A -85,B 0,C 180,E1 -1877.686,E2 -1877.686} C_VEL
LIN {X 0,Y 580.771,Z 463.043,A -85,B 0,C 180,E1 -1877.885,E2 -1877.885} C_VEL
LIN {X 0,Y 580.68,Z 474.292,A -85,B 0,C 180,E1 -1878.215,E2 -1878.215} C_VEL
LIN {X 0,Y 580.658,Z 483.459,A -85,B 0,C 180,E1 -1878.569,E2 -1878.569} C_VEL
LIN {X 0,Y 580.543,Z 494.139,A -85,B 0,C 180,E1 -1879.096,E2 -1879.096} C_VEL
LIN {X 0,Y 580.41,Z 504.128,A -85,B 0,C 180,E1 -1879.712,E2 -1879.712} C_VEL
LIN {X 0,Y 580.361,Z 513.464,A -85,B 0,C 180,E1 -1880.415,E2 -1880.415} C_VEL
LIN {X 0,Y 580.305,Z 521.289,A -85,B 0,C 180,E1 -1881.117,E2 -1881.117} C_VEL
LIN {X 0,Y 580.236,Z 529.412,A -85,B 0,C 180,E1 -1881.993,E2 -1881.993} C_VEL
LIN {X 0,Y 580.182,Z 536.179,A -85,B 0,C 180,E1 -1882.868,E2 -1882.868} C_VEL
LIN {X 0,Y 580.143,Z 541.837,A -85,B 0,C 180,E1 -1883.741,E2 -1883.741} C_VEL
LIN {X 0,Y 580.08,Z 547.325,A -85,B 0,C 180,E1 -1884.786,E2 -1884.786} C_VEL
LIN {X 0,Y 580.101,Z 551.641,A -85,B 0,C 180,E1 -1885.831,E2 -1885.831} C_VEL
LIN {X 0,Y 580.116,Z 553.936,A -85,B 0,C 180,E1 -1886.527,E2 -1886.527} C_VEL
LIN {X 0,Y 580.032,Z 557.187,A -85,B 0,C 180,E1 -1887.917,E2 -1887.917} C_VEL
LIN {X 0,Y 580.033,Z 558.713,A -85,B 0,C 180,E1 -1889.306,E2 -1889.306} C_VEL
LIN {X 0,Y 580.031,Z 559,A -85,B 0,C 180,E1 -1890,E2 -1890} C_VEL
LIN {X 0,Y 580.036,Z 558.138,A -85,B 0,C 180,E1 -1891.389,E2 -1891.389} C_VEL
LIN {X 0,Y 580.032,Z 557.188,A -85,B 0,C 180,E1 -1892.083,E2 -1892.083} C_VEL
LIN {X 0,Y 580.116,Z 553.938,A -85,B 0,C 180,E1 -1893.473,E2 -1893.473} C_VEL
LIN {X 0,Y 580.104,Z 550.358,A -85,B 0,C 180,E1 -1894.517,E2 -1894.517} C_VEL
LIN {X 0,Y 580.132,Z 545.664,A -85,B 0,C 180,E1 -1895.562,E2 -1895.562} C_VEL
LIN {X 0,Y 580.166,Z 539.593,A -85,B 0,C 180,E1 -1896.625,E2 -1896.625} C_VEL
LIN {X 0,Y 580.197,Z 533.673,A -85,B 0,C 180,E1 -1897.482,E2 -1897.482} C_VEL
LIN {X 0,Y 580.246,Z 526.391,A -85,B 0,C 180,E1 -1898.357,E2 -1898.357} C_VEL
LIN {X 0,Y 580.331,Z 517.533,A -85,B 0,C 180,E1 -1899.234,E2 -1899.234} C_VEL
LIN {X 0,Y 580.401,Z 509.025,A -85,B 0,C 180,E1 -1899.936,E2 -1899.936} C_VEL
LIN {X 0,Y 580.485,Z 500.115,A -85,B 0,C 180,E1 -1900.551,E2 -1900.551} C_VEL
LIN {X 0,Y 580.596,Z 490.902,A -85,B 0,C 180,E1 -1901.079,E2 -1901.079} C_VEL
LIN {X 0,Y 580.666,Z 479.12,A -85,B 0,C 180,E1 -1901.608,E2 -1901.608} C_VEL
LIN {X 0,Y 580.753,Z 468.029,A -85,B 0,C 180,E1 -1901.983,E2 -1901.983} C_VEL
LIN {X 0,Y 580.822,Z 456.959,A -85,B 0,C 180,E1 -1902.247,E2 -1902.247} C_VEL
LIN {X 0,Y 580.831,Z 440.158,A -85,B 0,C 180,E1 -1902.491,E2 -1902.491} C_VEL
LIN {X 0,Y 580.77,Z 349.83,A -85,B 0,C 180,E1 -1903.615,E2 -1903.615} C_VEL
LIN {X 0,Y 580.402,Z 347.279,A -85,B 0,C 180,E1 -1903.68,E2 -1903.68} C_VEL
LIN {X 0,Y 580.496,Z 329.123,A -85,B 0,C 180,E1 -1906.349,E2 -1906.349} C_VEL
LIN {X 0,Y 580.611,Z 312.231,A -85,B 0,C 180,E1 -1908.893,E2 -1908.893} C_VEL
LIN {X 0,Y 580.834,Z 295.46,A -85,B 0,C 180,E1 -1911.452,E2 -1911.452} C_VEL
LIN {X 0,Y 580.312,Z 290.923,A -85,B 0,C 180,E1 -1912.191,E2 -1912.191} C_VEL
LIN {X 0,Y 580.263,Z 290.699,A -85,B 0,C 180,E1 -1914.718,E2 -1914.718} C_VEL
LIN {X 0,Y 580.241,Z 290.703,A -85,B 0,C 180,E1 -1917.404,E2 -1917.404} C_VEL
LIN {X 0,Y 580.262,Z 290.702,A -85,B 0,C 180,E1 -1919.774,E2 -1919.774} C_VEL
LIN {X 0,Y 580.295,Z 290.702,A -85,B 0,C 180,E1 -1922.201,E2 -1922.201} C_VEL
LIN {X 0,Y 580.283,Z 290.705,A -85,B 0,C 180,E1 -1924.697,E2 -1924.697} C_VEL
LIN {X 0,Y 580.294,Z 290.696,A -85,B 0,C 180,E1 -1927.269,E2 -1927.269} C_VEL
LIN {X 0,Y 580.288,Z 290.694,A -85,B 0,C 180,E1 -1930.27,E2 -1930.27} C_VEL
LIN {X 0,Y 580.263,Z 290.701,A -85,B 0,C 180,E1 -1932.708,E2 -1932.708} C_VEL
LIN {X 0,Y 580.266,Z 290.704,A -85,B 0,C 180,E1 -1935.61,E2 -1935.61} C_VEL
LIN {X 0,Y 580.297,Z 290.694,A -85,B 0,C 180,E1 -1938.233,E2 -1938.233} C_VEL
LIN {X 0,Y 580.276,Z 290.696,A -85,B 0,C 180,E1 -1940.965,E2 -1940.965} C_VEL
LIN {X 0,Y 580.271,Z 290.702,A -85,B 0,C 180,E1 -1943.597,E2 -1943.597} C_VEL
LIN {X 0,Y 580.316,Z 290.703,A -85,B 0,C 180,E1 -1946.146,E2 -1946.146} C_VEL
LIN {X 0,Y 580.286,Z 290.7,A -85,B 0,C 180,E1 -1948.615,E2 -1948.615} C_VEL
LIN {X 0,Y 580.294,Z 290.696,A -85,B 0,C 180,E1 -1951.024,E2 -1951.024} C_VEL
LIN {X 0,Y 580.292,Z 290.693,A -85,B 0,C 180,E1 -1953.666,E2 -1953.666} C_VEL
LIN {X 0,Y 580.299,Z 290.693,A -85,B 0,C 180,E1 -1955.684,E2 -1955.684} C_VEL
LIN {X 0,Y 580.286,Z 290.7,A -85,B 0,C 180,E1 -1958.695,E2 -1958.695} C_VEL
LIN {X 0,Y 580.321,Z 290.697,A -85,B 0,C 180,E1 -1960.914,E2 -1960.914} C_VEL
LIN {X 0,Y 580.281,Z 290.699,A -85,B 0,C 180,E1 -1963.826,E2 -1963.826} C_VEL
LIN {X 0,Y 580.329,Z 290.692,A -85,B 0,C 180,E1 -1965.983,E2 -1965.983} C_VEL
LIN {X 0,Y 580.307,Z 290.692,A -85,B 0,C 180,E1 -1968.827,E2 -1968.827} C_VEL
LIN {X 0,Y 580.337,Z 290.693,A -85,B 0,C 180,E1 -1971.644,E2 -1971.644} C_VEL
LIN {X 0,Y 580.325,Z 290.695,A -85,B 0,C 180,E1 -1974.44,E2 -1974.44} C_VEL
LIN {X 0,Y 580.344,Z 290.687,A -85,B 0,C 180,E1 -1977.224,E2 -1977.224} C_VEL
LIN {X 0,Y 580.357,Z 290.687,A -85,B 0,C 180,E1 -1980,E2 -1980} C_VEL
LIN {X 0,Y 580.343,Z 290.699,A -85,B 0,C 180,E1 -1982.777,E2 -1982.777} C_VEL
LIN {X 0,Y 580.328,Z 290.691,A -85,B 0,C 180,E1 -1985.56,E2 -1985.56} C_VEL
LIN {X 0,Y 580.336,Z 290.688,A -85,B 0,C 180,E1 -1988.356,E2 -1988.356} C_VEL
LIN {X 0,Y 580.303,Z 290.701,A -85,B 0,C 180,E1 -1991.191,E2 -1991.191} C_VEL
LIN {X 0,Y 580.32,Z 290.694,A -85,B 0,C 180,E1 -1994.017,E2 -1994.017} C_VEL
LIN {X 0,Y 580.315,Z 290.691,A -85,B 0,C 180,E1 -1996.914,E2 -1996.914} C_VEL
LIN {X 0,Y 580.287,Z 290.702,A -85,B 0,C 180,E1 -1999.823,E2 -1999.823} C_VEL
LIN {X 0,Y 580.285,Z 290.695,A -85,B 0,C 180,E1 -2001.334,E2 -2001.334} C_VEL
LIN {X 0,Y 579.587,Z 290.791,A -85,B 0,C 180,E1 -2001.914,E2 -2001.914} C_VEL
LIN {X 0,Y 576.709,Z 291.143,A -85,B 0,C 180,E1 -2002.853,E2 -2002.853} C_VEL
LIN {X 0,Y 574.314,Z 291.441,A -85,B 0,C 180,E1 -2003.61,E2 -2003.61} C_VEL
LIN {X 0,Y 573.316,Z 291.573,A -85,B 0,C 180,E1 -2004.193,E2 -2004.193} C_VEL
LIN {X 0,Y 573.251,Z 291.575,A -85,B 0,C 180,E1 -2004.391,E2 -2004.391} C_VEL
LIN {X 0,Y 573.205,Z 291.579,A -85,B 0,C 180,E1 -2006.978,E2 -2006.978} C_VEL
LIN {X 0,Y 573.244,Z 291.572,A -85,B 0,C 180,E1 -2009.487,E2 -2009.487} C_VEL
LIN {X 0,Y 573.254,Z 291.577,A -85,B 0,C 180,E1 -2012.645,E2 -2012.645} C_VEL
LIN {X 0,Y 573.205,Z 291.587,A -85,B 0,C 180,E1 -2015.188,E2 -2015.188} C_VEL
LIN {X 0,Y 573.232,Z 291.576,A -85,B 0,C 180,E1 -2017.808,E2 -2017.808} C_VEL
LIN {X 0,Y 573.246,Z 291.573,A -85,B 0,C 180,E1 -2020.525,E2 -2020.525} C_VEL
LIN {X 0,Y 573.239,Z 291.58,A -85,B 0,C 180,E1 -2023.359,E2 -2023.359} C_VEL
LIN {X 0,Y 573.259,Z 291.706,A -85,B 0,C 180,E1 -2025.322,E2 -2025.322} C_VEL
LIN {X 0,Y 573.658,Z 295.674,A -85,B 0,C 180,E1 -2026.036,E2 -2026.036} C_VEL
LIN {X 0,Y 573.484,Z 312.139,A -85,B 0,C 180,E1 -2028.799,E2 -2028.799} C_VEL
LIN {X 0,Y 573.325,Z 330.363,A -85,B 0,C 180,E1 -2031.814,E2 -2031.814} C_VEL
LIN {X 0,Y 573.335,Z 332.959,A -85,B 0,C 180,E1 -2032.2,E2 -2032.2} C_VEL
LIN {X 0,Y 574.059,Z 337.83,A -85,B 0,C 180,E1 -2032.305,E2 -2032.305} C_VEL
LIN {X 0,Y 573.877,Z 438.612,A -85,B 0,C 180,E1 -2033.589,E2 -2033.589} C_VEL
LIN {X 0,Y 573.801,Z 448.374,A -85,B 0,C 180,E1 -2033.789,E2 -2033.789} C_VEL
LIN {X 0,Y 573.734,Z 458.728,A -85,B 0,C 180,E1 -2034.095,E2 -2034.095} C_VEL
LIN {X 0,Y 573.677,Z 469.494,A -85,B 0,C 180,E1 -2034.523,E2 -2034.523} C_VEL
LIN {X 0,Y 573.556,Z 479.844,A -85,B 0,C 180,E1 -2035.049,E2 -2035.049} C_VEL
LIN {X 0,Y 573.416,Z 489.84,A -85,B 0,C 180,E1 -2035.682,E2 -2035.682} C_VEL
LIN {X 0,Y 573.373,Z 498.142,A -85,B 0,C 180,E1 -2036.314,E2 -2036.314} C_VEL
LIN {X 0,Y 573.292,Z 506.206,A -85,B 0,C 180,E1 -2037.044,E2 -2037.044} C_VEL
LIN {X 0,Y 573.17,Z 514.757,A -85,B 0,C 180,E1 -2037.982,E2 -2037.982} C_VEL
LIN {X 0,Y 573.101,Z 520.981,A -85,B 0,C 180,E1 -2038.794,E2 -2038.794} C_VEL
LIN {X 0,Y 573.077,Z 527.413,A -85,B 0,C 180,E1 -2039.814,E2 -2039.814} C_VEL
LIN {X 0,Y 573.044,Z 531.698,A -85,B 0,C 180,E1 -2040.622,E2 -2040.622} C_VEL
LIN {X 0,Y 573.009,Z 536.403,A -85,B 0,C 180,E1 -2041.752,E2 -2041.752} C_VEL
LIN {X 0,Y 572.986,Z 539.218,A -85,B 0,C 180,E1 -2042.616,E2 -2042.616} C_VEL
LIN {X 0,Y 572.945,Z 541.966,A -85,B 0,C 180,E1 -2043.795,E2 -2043.795} C_VEL
LIN {X 0,Y 572.905,Z 543.647,A -85,B 0,C 180,E1 -2045.2,E2 -2045.2} C_VEL
LIN {X 0,Y 572.915,Z 543.989,A -85,B 0,C 180,E1 -2046.121,E2 -2046.121} C_VEL
LIN {X 0,Y 572.951,Z 543.632,A -85,B 0,C 180,E1 -2046.922,E2 -2046.922} C_VEL
LIN {X 0,Y 572.941,Z 541.729,A -85,B 0,C 180,E1 -2048.408,E2 -2048.408} C_VEL
LIN {X 0,Y 572.989,Z 539.008,A -85,B 0,C 180,E1 -2049.539,E2 -2049.539} C_VEL
LIN {X 0,Y 572.995,Z 534.532,A -85,B 0,C 180,E1 -2050.81,E2 -2050.81} C_VEL
LIN {X 0,Y 573.05,Z 530.121,A -85,B 0,C 180,E1 -2051.776,E2 -2051.776} C_VEL
LIN {X 0,Y 573.109,Z 524.935,A -85,B 0,C 180,E1 -2052.7,E2 -2052.7} C_VEL
LIN {X 0,Y 573.148,Z 518.677,A -85,B 0,C 180,E1 -2053.619,E2 -2053.619} C_VEL
LIN {X 0,Y 573.188,Z 511.129,A -85,B 0,C 180,E1 -2054.533,E2 -2054.533} C_VEL
LIN {X 0,Y 573.323,Z 502.682,A -85,B 0,C 180,E1 -2055.379,E2 -2055.379} C_VEL
LIN {X 0,Y 573.412,Z 494.319,A -85,B 0,C 180,E1 -2056.082,E2 -2056.082} C_VEL
LIN {X 0,Y 573.503,Z 485.282,A -85,B 0,C 180,E1 -2056.716,E2 -2056.716} C_VEL
LIN {X 0,Y 573.605,Z 475.934,A -85,B 0,C 180,E1 -2057.259,E2 -2057.259} C_VEL
LIN {X 0,Y 573.722,Z 463.971,A -85,B 0,C 180,E1 -2057.801,E2 -2057.801} C_VEL
LIN {X 0,Y 573.834,Z 453.546,A -85,B 0,C 180,E1 -2058.16,E2 -2058.16} C_VEL
LIN {X 0,Y 573.888,Z 442.295,A -85,B 0,C 180,E1 -2058.437,E2 -2058.437} C_VEL
LIN {X 0,Y 573.933,Z 425.563,A -85,B 0,C 180,E1 -2058.683,E2 -2058.683} C_VEL
LIN {X 0,Y 573.991,Z 337.094,A -85,B 0,C 180,E1 -2059.796,E2 -2059.796} C_VEL
LIN {X 0,Y 573.385,Z 333.199,A -85,B 0,C 180,E1 -2059.874,E2 -2059.874} C_VEL
LIN {X 0,Y 573.322,Z 331.325,A -85,B 0,C 180,E1 -2060.118,E2 -2060.118} C_VEL
LIN {X 0,Y 573.476,Z 315.182,A -85,B 0,C 180,E1 -2062.784,E2 -2062.784} C_VEL
LIN {X 0,Y 573.651,Z 296.23,A -85,B 0,C 180,E1 -2065.96,E2 -2065.96} C_VEL
LIN {X 0,Y 573.322,Z 291.758,A -85,B 0,C 180,E1 -2066.75,E2 -2066.75} C_VEL
LIN {X 0,Y 573.329,Z 291.562,A -85,B 0,C 180,E1 -2069.298,E2 -2069.298} C_VEL
LIN {X 0,Y 573.308,Z 291.567,A -85,B 0,C 180,E1 -2072.108,E2 -2072.108} C_VEL
LIN {X 0,Y 573.291,Z 291.567,A -85,B 0,C 180,E1 -2075.628,E2 -2075.628} C_VEL
LIN {X 0,Y 573.274,Z 291.57,A -85,B 0,C 180,E1 -2077.75,E2 -2077.75} C_VEL
LIN {X 0,Y 573.268,Z 291.569,A -85,B 0,C 180,E1 -2080.597,E2 -2080.597} C_VEL
LIN {X 0,Y 573.266,Z 291.568,A -85,B 0,C 180,E1 -2082.749,E2 -2082.749} C_VEL
LIN {X 0,Y 573.236,Z 291.572,A -85,B 0,C 180,E1 -2084.92,E2 -2084.92} C_VEL
LIN {X 0,Y 573.253,Z 291.578,A -85,B 0,C 180,E1 -2087.848,E2 -2087.848} C_VEL
LIN {X 0,Y 573.246,Z 291.578,A -85,B 0,C 180,E1 -2090.077,E2 -2090.077} C_VEL
LIN {X 0,Y 573.235,Z 291.582,A -85,B 0,C 180,E1 -2092.338,E2 -2092.338} C_VEL
LIN {X 0,Y 573.247,Z 291.572,A -85,B 0,C 180,E1 -2095.411,E2 -2095.411} C_VEL
LIN {X 0,Y 573.253,Z 291.569,A -85,B 0,C 180,E1 -2098.029,E2 -2098.029} C_VEL
LIN {X 0,Y 573.231,Z 291.578,A -85,B 0,C 180,E1 -2100.882,E2 -2100.882} C_VEL
LIN {X 0,Y 573.265,Z 291.578,A -85,B 0,C 180,E1 -2103.524,E2 -2103.524} C_VEL
LIN {X 0,Y 573.195,Z 291.582,A -85,B 0,C 180,E1 -2106.053,E2 -2106.053} C_VEL
LIN {X 0,Y 573.239,Z 291.572,A -85,B 0,C 180,E1 -2108.702,E2 -2108.702} C_VEL
LIN {X 0,Y 573.23,Z 291.573,A -85,B 0,C 180,E1 -2111.593,E2 -2111.593} C_VEL
LIN {X 0,Y 573.23,Z 291.583,A -85,B 0,C 180,E1 -2114.334,E2 -2114.334} C_VEL
LIN {X 0,Y 573.227,Z 291.574,A -85,B 0,C 180,E1 -2117.36,E2 -2117.36} C_VEL
LIN {X 0,Y 573.24,Z 291.571,A -85,B 0,C 180,E1 -2120.392,E2 -2120.392} C_VEL
LIN {X 0,Y 573.254,Z 291.579,A -85,B 0,C 180,E1 -2123.078,E2 -2123.078} C_VEL
LIN {X 0,Y 573.256,Z 291.576,A -85,B 0,C 180,E1 -2125.67,E2 -2125.67} C_VEL
LIN {X 0,Y 573.241,Z 291.572,A -85,B 0,C 180,E1 -2128.184,E2 -2128.184} C_VEL
LIN {X 0,Y 573.261,Z 291.565,A -85,B 0,C 180,E1 -2130.634,E2 -2130.634} C_VEL
LIN {X 0,Y 573.212,Z 291.576,A -85,B 0,C 180,E1 -2133.513,E2 -2133.513} C_VEL
LIN {X 0,Y 573.229,Z 291.581,A -85,B 0,C 180,E1 -2136.134,E2 -2136.134} C_VEL
LIN {X 0,Y 573.248,Z 291.571,A -85,B 0,C 180,E1 -2139.173,E2 -2139.173} C_VEL
LIN {X 0,Y 573.209,Z 291.572,A -85,B 0,C 180,E1 -2141.411,E2 -2141.411} C_VEL
LIN {X 0,Y 573.236,Z 291.571,A -85,B 0,C 180,E1 -2143.621,E2 -2143.621} C_VEL
LIN {X 0,Y 573.221,Z 291.575,A -85,B 0,C 180,E1 -2146.529,E2 -2146.529} C_VEL
LIN {X 0,Y 573.251,Z 291.581,A -85,B 0,C 180,E1 -2149.403,E2 -2149.403} C_VEL
LIN {X 0,Y 573.219,Z 291.573,A -85,B 0,C 180,E1 -2152.249,E2 -2152.249} C_VEL
LIN {X 0,Y 573.29,Z 291.562,A -85,B 0,C 180,E1 -2155.077,E2 -2155.077} C_VEL
LIN {X 0,Y 573.309,Z 291.568,A -85,B 0,C 180,E1 -2157.892,E2 -2157.892} C_VEL
LIN {X 0,Y 573.329,Z 291.567,A -85,B 0,C 180,E1 -2160.702,E2 -2160.702} C_VEL
LIN {X 0,Y 573.297,Z 291.571,A -85,B 0,C 180,E1 -2162.81,E2 -2162.81} C_VEL
LIN {X 0,Y 573.268,Z 291.566,A -85,B 0,C 180,E1 -2165.628,E2 -2165.628} C_VEL
LIN {X 0,Y 573.221,Z 291.575,A -85,B 0,C 180,E1 -2167.751,E2 -2167.751} C_VEL
LIN {X 0,Y 573.239,Z 291.573,A -85,B 0,C 180,E1 -2170.597,E2 -2170.597} C_VEL
LIN {X 0,Y 573.202,Z 291.586,A -85,B 0,C 180,E1 -2173.471,E2 -2173.471} C_VEL
LIN {X 0,Y 573.203,Z 291.578,A -85,B 0,C 180,E1 -2176.379,E2 -2176.379} C_VEL
LIN {X 0,Y 573.267,Z 291.569,A -85,B 0,C 180,E1 -2179.33,E2 -2179.33} C_VEL
